  Set speed (76.2 mm/s)
  MoveL 645 to (-197.85, 148.44, -8.4) mm, rotated rx -174.06 ry -29.54 rz -11.91 deg; joints [4.931, -49.184, 110.878, -80.007, 60.979, 152.328]
  MoveL 646 to (-199.6, 148.44, -8.41) mm, rotated rx -174.06 ry -29.54 rz -11.91 deg; joints [4.86, -49.19, 110.892, -80.07, 60.944, 152.33]
  MoveL 647 to (-206.05, 148.44, -11.57) mm, rotated rx -174.06 ry -29.54 rz -11.91 deg; joints [4.602, -49.043, 110.941, -80.393, 60.791, 152.527]
  MoveL 648 to (-201.08, 148.44, -20.25) mm, rotated rx -174.06 ry -29.54 rz -11.91 deg; joints [4.803, -48.562, 110.904, -80.469, 60.81, 153.047]
  MoveL 649 to (-201.08, 145.27, -20.25) mm, rotated rx -174.06 ry -29.54 rz -11.91 deg; joints [4.814, -48.698, 111.183, -80.539, 60.791, 153.21]
  MoveL 650 to (-206.05, 145.27, -11.57) mm, rotated rx -174.06 ry -29.54 rz -11.91 deg; joints [4.613, -49.18, 111.22, -80.463, 60.772, 152.689]
  MoveL 651 to (-199.6, 145.27, -8.41) mm, rotated rx -174.06 ry -29.54 rz -11.91 deg; joints [4.872, -49.327, 111.171, -80.138, 60.925, 152.491]
  MoveL 652 to (-197.85, 145.27, -8.4) mm, rotated rx -174.06 ry -29.54 rz -11.91 deg; joints [4.942, -49.321, 111.158, -80.075, 60.959, 152.489]
  MoveL 653 to (-197.85, 145.27, -4.14) mm, rotated rx -174.06 ry -29.54 rz -11.91 deg; joints [4.941, -49.548, 111.154, -79.95, 60.999, 152.23]
  Set speed (38.1 mm/s)
  MoveL 654 to (-197.89, 145.27, -3.98) mm, rotated rx -174.06 ry -29.54 rz -11.91 deg; joints [4.939, -49.557, 111.155, -79.947, 60.999, 152.22]
  MoveL 655 to (-198.05, 144.95, -3.7) mm, rotated rx -174.06 ry -29.54 rz -11.91 deg; joints [4.934, -49.585, 111.183, -79.951, 60.997, 152.22]
  Set speed (76.2 mm/s)
  MoveL 656 to (-198.05, 142.41, -3.7) mm, rotated rx -174.06 ry -29.54 rz -11.91 deg; joints [4.943, -49.696, 111.406, -80.005, 60.981, 152.347]
  Set speed (38.1 mm/s)
  MoveL 657 to (-197.89, 142.09, -3.98) mm, rotated rx -174.06 ry -29.54 rz -11.91 deg; joints [4.951, -49.694, 111.433, -80.014, 60.98, 152.38]
  MoveL 658 to (-197.85, 142.09, -4.14) mm, rotated rx -174.06 ry -29.54 rz -11.91 deg; joints [4.952, -49.686, 111.433, -80.017, 60.979, 152.39]
  Set speed (76.2 mm/s)
  MoveL 659 to (-197.85, 142.09, -8.4) mm, rotated rx -174.06 ry -29.54 rz -11.91 deg; joints [4.953, -49.458, 111.436, -80.143, 60.94, 152.65]
  MoveL 660 to (-199.6, 142.09, -8.41) mm, rotated rx -174.06 ry -29.54 rz -11.91 deg; joints [4.883, -49.464, 111.45, -80.206, 60.906, 152.652]
  MoveL 661 to (-206.05, 142.09, -11.57) mm, rotated rx -174.06 ry -29.54 rz -11.91 deg; joints [4.623, -49.316, 111.499, -80.533, 60.753, 152.851]
  MoveL 662 to (-201.08, 142.09, -20.25) mm, rotated rx -174.06 ry -29.54 rz -11.91 deg; joints [4.825, -48.833, 111.462, -80.609, 60.773, 153.374]
  MoveL 663 to (-201.08, 138.92, -20.25) mm, rotated rx -174.06 ry -29.54 rz -11.91 deg; joints [4.836, -48.967, 111.74, -80.678, 60.754, 153.537]
  MoveL 664 to (-206.05, 138.92, -11.57) mm, rotated rx -174.06 ry -29.54 rz -11.91 deg; joints [4.634, -49.453, 111.777, -80.602, 60.735, 153.012]
  MoveL 665 to (-199.6, 138.92, -8.41) mm, rotated rx -174.06 ry -29.54 rz -11.91 deg; joints [4.894, -49.6, 111.728, -80.275, 60.887, 152.813]
  MoveL 666 to (-197.85, 138.92, -8.4) mm, rotated rx -174.06 ry -29.54 rz -11.91 deg; joints [4.965, -49.595, 111.714, -80.211, 60.921, 152.81]
  MoveL 667 to (-197.85, 138.92, -4.14) mm, rotated rx -174.06 ry -29.54 rz -11.91 deg; joints [4.964, -49.823, 111.711, -80.085, 60.96, 152.549]
  Set speed (38.1 mm/s)
  MoveL 668 to (-197.89, 138.92, -3.98) mm, rotated rx -174.06 ry -29.54 rz -11.91 deg; joints [4.962, -49.832, 111.711, -80.082, 60.961, 152.54]
  MoveL 669 to (-198.05, 138.6, -3.7) mm, rotated rx -174.06 ry -29.54 rz -11.91 deg; joints [4.957, -49.861, 111.74, -80.086, 60.959, 152.539]
  Set speed (76.2 mm/s)
  MoveL 670 to (-198.05, 136.06, -3.7) mm, rotated rx -174.06 ry -29.54 rz -11.91 deg; joints [4.966, -49.97, 111.962, -80.14, 60.944, 152.666]
  Set speed (38.1 mm/s)
  MoveL 671 to (-197.89, 135.74, -3.98) mm, rotated rx -174.06 ry -29.54 rz -11.91 deg; joints [4.973, -49.969, 111.989, -80.149, 60.942, 152.699]
  MoveL 672 to (-197.85, 135.74, -4.14) mm, rotated rx -174.06 ry -29.54 rz -11.91 deg; joints [4.975, -49.96, 111.988, -80.152, 60.942, 152.709]
  Set speed (76.2 mm/s)
  MoveL 673 to (-197.85, 135.74, -8.4) mm, rotated rx -174.06 ry -29.54 rz -11.91 deg; joints [4.976, -49.731, 111.992, -80.279, 60.903, 152.971]
  MoveL 674 to (-199.6, 135.74, -8.41) mm, rotated rx -174.06 ry -29.54 rz -11.91 deg; joints [4.905, -49.737, 112.005, -80.343, 60.869, 152.973]
  MoveL 675 to (-206.05, 135.74, -11.57) mm, rotated rx -174.06 ry -29.54 rz -11.91 deg; joints [4.644, -49.588, 112.055, -80.671, 60.717, 153.173]
  MoveL 676 to (-201.08, 135.74, -20.25) mm, rotated rx -174.06 ry -29.54 rz -11.91 deg; joints [4.848, -49.102, 112.018, -80.748, 60.736, 153.699]
  MoveL 677 to (-201.08, 132.57, -20.25) mm, rotated rx -174.06 ry -29.54 rz -11.91 deg; joints [4.859, -49.236, 112.295, -80.818, 60.718, 153.862]
  MoveL 678 to (-206.05, 132.57, -11.57) mm, rotated rx -174.06 ry -29.54 rz -11.91 deg; joints [4.655, -49.724, 112.332, -80.741, 60.699, 153.334]
  MoveL 679 to (-199.6, 132.57, -8.41) mm, rotated rx -174.06 ry -29.54 rz -11.91 deg; joints [4.916, -49.873, 112.282, -80.411, 60.85, 153.133]
  MoveL 680 to (-197.85, 132.57, -8.4) mm, rotated rx -174.06 ry -29.54 rz -11.91 deg; joints [4.987, -49.867, 112.269, -80.346, 60.884, 153.13]
  MoveL 681 to (-197.85, 132.57, -4.14) mm, rotated rx -174.06 ry -29.54 rz -11.91 deg; joints [4.987, -50.097, 112.265, -80.219, 60.923, 152.868]
  Set speed (38.1 mm/s)
  MoveL 682 to (-197.89, 132.57, -3.98) mm, rotated rx -174.06 ry -29.54 rz -11.91 deg; joints [4.985, -50.105, 112.266, -80.216, 60.924, 152.858]
  MoveL 683 to (-198.05, 132.25, -3.7) mm, rotated rx -174.06 ry -29.54 rz -11.91 deg; joints [4.979, -50.135, 112.294, -80.22, 60.921, 152.857]
  Set speed (76.2 mm/s)
  MoveL 684 to (-198.05, 129.71, -3.7) mm, rotated rx -174.06 ry -29.54 rz -11.91 deg; joints [4.989, -50.244, 112.515, -80.274, 60.906, 152.984]
  Set speed (38.1 mm/s)
  MoveL 685 to (-197.89, 129.39, -3.98) mm, rotated rx -174.06 ry -29.54 rz -11.91 deg; joints [4.996, -50.242, 112.542, -80.283, 60.905, 153.017]
  MoveL 686 to (-197.85, 129.39, -4.14) mm, rotated rx -174.06 ry -29.54 rz -11.91 deg; joints [4.998, -50.233, 112.542, -80.286, 60.905, 153.026]
  Set speed (76.2 mm/s)
  MoveL 687 to (-197.85, 129.39, -8.4) mm, rotated rx -174.06 ry -29.54 rz -11.91 deg; joints [4.999, -50.003, 112.545, -80.414, 60.866, 153.29]
  MoveL 688 to (-199.6, 129.39, -8.41) mm, rotated rx -174.06 ry -29.54 rz -11.91 deg; joints [4.928, -50.009, 112.559, -80.478, 60.832, 153.293]
  MoveL 689 to (-206.05, 129.39, -11.57) mm, rotated rx -174.06 ry -29.54 rz -11.91 deg; joints [4.666, -49.859, 112.608, -80.81, 60.681, 153.495]
  MoveL 690 to (-201.08, 129.39, -20.25) mm, rotated rx -174.06 ry -29.54 rz -11.91 deg; joints [4.87, -49.37, 112.571, -80.887, 60.701, 154.024]
  MoveL 691 to (-201.08, 126.22, -20.25) mm, rotated rx -174.06 ry -29.54 rz -11.91 deg; joints [4.881, -49.504, 112.847, -80.956, 60.683, 154.186]
  MoveL 692 to (-206.05, 126.22, -11.57) mm, rotated rx -174.06 ry -29.54 rz -11.91 deg; joints [4.677, -49.994, 112.884, -80.879, 60.664, 153.655]
  MoveL 693 to (-199.6, 126.22, -8.41) mm, rotated rx -174.06 ry -29.54 rz -11.91 deg; joints [4.939, -50.144, 112.834, -80.546, 60.814, 153.452]
  MoveL 694 to (-197.85, 126.22, -8.4) mm, rotated rx -174.06 ry -29.54 rz -11.91 deg; joints [5.01, -50.138, 112.821, -80.481, 60.848, 153.45]
  MoveL 695 to (-197.85, 126.22, -4.14) mm, rotated rx -174.06 ry -29.54 rz -11.91 deg; joints [5.01, -50.37, 112.818, -80.353, 60.886, 153.185]
  Set speed (38.1 mm/s)
  MoveL 696 to (-197.89, 126.22, -3.98) mm, rotated rx -174.06 ry -29.54 rz -11.91 deg; joints [5.008, -50.378, 112.818, -80.35, 60.887, 153.175]
  MoveL 697 to (-198.05, 125.9, -3.7) mm, rotated rx -174.06 ry -29.54 rz -11.91 deg; joints [5.002, -50.407, 112.846, -80.354, 60.885, 153.174]
  Set speed (76.2 mm/s)
  MoveL 698 to (-198.05, 123.36, -3.7) mm, rotated rx -174.06 ry -29.54 rz -11.91 deg; joints [5.012, -50.516, 113.067, -80.408, 60.87, 153.301]
  Set speed (38.1 mm/s)
  MoveL 699 to (-197.89, 123.04, -3.98) mm, rotated rx -174.06 ry -29.54 rz -11.91 deg; joints [5.019, -50.514, 113.093, -80.417, 60.869, 153.333]
  MoveL 700 to (-197.85, 123.04, -4.14) mm, rotated rx -174.06 ry -29.54 rz -11.91 deg; joints [5.021, -50.506, 113.093, -80.42, 60.868, 153.343]
  Set speed (76.2 mm/s)
  MoveL 701 to (-197.85, 123.04, -8.4) mm, rotated rx -174.06 ry -29.54 rz -11.91 deg; joints [5.022, -50.274, 113.096, -80.549, 60.83, 153.609]
  MoveL 702 to (-199.6, 123.04, -8.41) mm, rotated rx -174.06 ry -29.54 rz -11.91 deg; joints [4.95, -50.28, 113.11, -80.614, 60.796, 153.611]
  MoveL 703 to (-206.05, 123.04, -11.57) mm, rotated rx -174.06 ry -29.54 rz -11.91 deg; joints [4.687, -50.129, 113.159, -80.948, 60.646, 153.816]
  MoveL 704 to (-201.08, 123.04, -20.25) mm, rotated rx -174.06 ry -29.54 rz -11.91 deg; joints [4.892, -49.637, 113.122, -81.025, 60.666, 154.348]
  MoveL 705 to (-201.08, 119.87, -20.25) mm, rotated rx -174.06 ry -29.54 rz -11.91 deg; joints [4.904, -49.77, 113.397, -81.094, 60.649, 154.509]
  MoveL 706 to (-206.05, 119.87, -11.57) mm, rotated rx -174.06 ry -29.54 rz -11.91 deg; joints [4.698, -50.264, 113.434, -81.016, 60.629, 153.975]
  MoveL 707 to (-199.6, 119.87, -8.41) mm, rotated rx -174.06 ry -29.54 rz -11.91 deg; joints [4.962, -50.415, 113.385, -80.681, 60.779, 153.77]
  MoveL 708 to (-197.85, 119.87, -8.4) mm, rotated rx -174.06 ry -29.54 rz -11.91 deg; joints [5.034, -50.409, 113.371, -80.616, 60.812, 153.768]
  MoveL 709 to (-197.85, 119.87, -4.14) mm, rotated rx -174.06 ry -29.54 rz -11.91 deg; joints [5.033, -50.641, 113.368, -80.487, 60.851, 153.501]
  Set speed (38.1 mm/s)
  MoveL 710 to (-197.89, 119.87, -3.98) mm, rotated rx -174.06 ry -29.54 rz -11.91 deg; joints [5.031, -50.65, 113.368, -80.483, 60.851, 153.491]
  MoveL 711 to (-198.05, 119.55, -3.7) mm, rotated rx -174.06 ry -29.54 rz -11.91 deg; joints [5.026, -50.679, 113.396, -80.488, 60.849, 153.49]
  Set speed (76.2 mm/s)
  MoveL 712 to (-198.05, 117.01, -3.7) mm, rotated rx -174.06 ry -29.54 rz -11.91 deg; joints [5.035, -50.788, 113.616, -80.541, 60.835, 153.616]
  Set speed (38.1 mm/s)
  MoveL 713 to (-197.89, 116.7, -3.98) mm, rotated rx -174.06 ry -29.54 rz -11.91 deg; joints [5.043, -50.786, 113.642, -80.55, 60.834, 153.649]
  MoveL 714 to (-197.85, 116.7, -4.14) mm, rotated rx -174.06 ry -29.54 rz -11.91 deg; joints [5.044, -50.777, 113.642, -80.553, 60.833, 153.659]
  Set speed (76.2 mm/s)
  MoveL 715 to (-197.85, 116.7, -8.4) mm, rotated rx -174.06 ry -29.54 rz -11.91 deg; joints [5.045, -50.543, 113.645, -80.683, 60.795, 153.926]
  MoveL 716 to (-199.6, 116.7, -8.41) mm, rotated rx -174.06 ry -29.54 rz -11.91 deg; joints [4.973, -50.549, 113.659, -80.748, 60.761, 153.929]
  MoveL 717 to (-206.05, 116.7, -11.57) mm, rotated rx -174.06 ry -29.54 rz -11.91 deg; joints [4.709, -50.398, 113.708, -81.085, 60.612, 154.135]
  MoveL 718 to (-201.08, 116.7, -20.25) mm, rotated rx -174.06 ry -29.54 rz -11.91 deg; joints [4.915, -49.903, 113.671, -81.163, 60.632, 154.671]
  MoveL 719 to (-201.08, 113.52, -20.25) mm, rotated rx -174.06 ry -29.54 rz -11.91 deg; joints [4.927, -50.035, 113.945, -81.232, 60.615, 154.832]
  MoveL 720 to (-206.05, 113.52, -11.57) mm, rotated rx -174.06 ry -29.54 rz -11.91 deg; joints [4.72, -50.532, 113.982, -81.153, 60.595, 154.295]
  MoveL 721 to (-199.6, 113.52, -8.41) mm, rotated rx -174.06 ry -29.54 rz -11.91 deg; joints [4.985, -50.684, 113.933, -80.815, 60.744, 154.088]
  MoveL 722 to (-197.85, 113.52, -8.4) mm, rotated rx -174.06 ry -29.54 rz -11.91 deg; joints [5.057, -50.678, 113.919, -80.75, 60.778, 154.085]
  MoveL 723 to (-197.85, 113.52, -4.14) mm, rotated rx -174.06 ry -29.54 rz -11.91 deg; joints [5.056, -50.912, 113.916, -80.62, 60.816, 153.817]
  Set speed (38.1 mm/s)
  MoveL 724 to (-197.89, 113.52, -3.98) mm, rotated rx -174.06 ry -29.54 rz -11.91 deg; joints [5.054, -50.921, 113.916, -80.616, 60.816, 153.807]
  MoveL 725 to (-198.05, 113.2, -3.7) mm, rotated rx -174.06 ry -29.54 rz -11.91 deg; joints [5.049, -50.95, 113.944, -80.62, 60.814, 153.805]
  Set speed (76.2 mm/s)
  MoveL 726 to (-198.05, 110.66, -3.7) mm, rotated rx -174.06 ry -29.54 rz -11.91 deg; joints [5.058, -51.058, 114.163, -80.673, 60.8, 153.931]
  Set speed (38.1 mm/s)
  MoveL 727 to (-197.89, 110.35, -3.98) mm, rotated rx -174.06 ry -29.54 rz -11.91 deg; joints [5.066, -51.056, 114.189, -80.682, 60.799, 153.964]
  MoveL 728 to (-197.85, 110.35, -4.14) mm, rotated rx -174.06 ry -29.54 rz -11.91 deg; joints [5.068, -51.047, 114.189, -80.686, 60.798, 153.974]
  Set speed (76.2 mm/s)
  MoveL 729 to (-197.85, 110.35, -8.4) mm, rotated rx -174.06 ry -29.54 rz -11.91 deg; joints [5.069, -50.812, 114.192, -80.816, 60.761, 154.243]
  MoveL 730 to (-199.6, 110.35, -8.41) mm, rotated rx -174.06 ry -29.54 rz -11.91 deg; joints [4.997, -50.818, 114.206, -80.882, 60.727, 154.246]
  MoveL 731 to (-206.05, 110.35, -11.57) mm, rotated rx -174.06 ry -29.54 rz -11.91 deg; joints [4.731, -50.665, 114.255, -81.222, 60.579, 154.454]
  MoveL 732 to (-201.08, 110.35, -20.25) mm, rotated rx -174.06 ry -29.54 rz -11.91 deg; joints [4.938, -50.167, 114.218, -81.301, 60.599, 154.993]
  MoveL 733 to (-201.08, 107.17, -20.25) mm, rotated rx -174.06 ry -29.54 rz -11.91 deg; joints [4.95, -50.299, 114.491, -81.369, 60.583, 155.153]
  MoveL 734 to (-206.05, 107.17, -11.57) mm, rotated rx -174.06 ry -29.54 rz -11.91 deg; joints [4.742, -50.799, 114.528, -81.29, 60.563, 154.613]
  MoveL 735 to (-199.6, 107.17, -8.41) mm, rotated rx -174.06 ry -29.54 rz -11.91 deg; joints [5.008, -50.952, 114.479, -80.949, 60.711, 154.404]
  MoveL 736 to (-197.85, 107.17, -8.4) mm, rotated rx -174.06 ry -29.54 rz -11.91 deg; joints [5.081, -50.946, 114.465, -80.883, 60.744, 154.401]
  MoveL 737 to (-197.85, 107.17, -4.14) mm, rotated rx -174.06 ry -29.54 rz -11.91 deg; joints [5.08, -51.181, 114.462, -80.752, 60.781, 154.131]
  Set speed (38.1 mm/s)
  MoveL 738 to (-197.89, 107.17, -3.98) mm, rotated rx -174.06 ry -29.54 rz -11.91 deg; joints [5.078, -51.19, 114.462, -80.749, 60.782, 154.121]
  MoveL 739 to (-198.05, 106.85, -3.7) mm, rotated rx -174.06 ry -29.54 rz -11.91 deg; joints [5.073, -51.22, 114.49, -80.753, 60.78, 154.12]
  Set speed (76.2 mm/s)
  MoveL 740 to (-198.05, 104.31, -3.7) mm, rotated rx -174.06 ry -29.54 rz -11.91 deg; joints [5.082, -51.327, 114.708, -80.805, 60.766, 154.245]
  Set speed (38.1 mm/s)
  MoveL 741 to (-197.89, 104, -3.98) mm, rotated rx -174.06 ry -29.54 rz -11.91 deg; joints [5.09, -51.325, 114.734, -80.814, 60.765, 154.278]
  MoveL 742 to (-197.85, 104, -4.14) mm, rotated rx -174.06 ry -29.54 rz -11.91 deg; joints [5.092, -51.316, 114.734, -80.818, 60.765, 154.288]
  Set speed (76.2 mm/s)
  MoveL 743 to (-197.85, 104, -8.4) mm, rotated rx -174.06 ry -29.54 rz -11.91 deg; joints [5.093, -51.08, 114.737, -80.949, 60.727, 154.559]
  MoveL 744 to (-199.6, 104, -8.41) mm, rotated rx -174.06 ry -29.54 rz -11.91 deg; joints [5.02, -51.086, 114.751, -81.016, 60.694, 154.562]
  MoveL 745 to (-206.05, 104, -11.57) mm, rotated rx -174.06 ry -29.54 rz -11.91 deg; joints [4.753, -50.932, 114.801, -81.358, 60.546, 154.772]
  MoveL 746 to (-201.08, 104, -20.25) mm, rotated rx -174.06 ry -29.54 rz -11.91 deg; joints [4.961, -50.431, 114.763, -81.438, 60.567, 155.314]
  MoveL 747 to (-201.08, 100.82, -20.25) mm, rotated rx -174.06 ry -29.54 rz -11.91 deg; joints [4.973, -50.562, 115.035, -81.506, 60.551, 155.474]
  MoveL 748 to (-206.05, 100.82, -11.57) mm, rotated rx -174.06 ry -29.54 rz -11.91 deg; joints [4.765, -51.065, 115.072, -81.426, 60.53, 154.93]
  MoveL 749 to (-199.6, 100.82, -8.41) mm, rotated rx -174.06 ry -29.54 rz -11.91 deg; joints [5.032, -51.219, 115.023, -81.082, 60.678, 154.72]
  MoveL 750 to (-197.85, 100.82, -8.4) mm, rotated rx -174.06 ry -29.54 rz -11.91 deg; joints [5.105, -51.213, 115.009, -81.016, 60.711, 154.716]
  MoveL 751 to (-197.85, 100.82, -4.14) mm, rotated rx -174.06 ry -29.54 rz -11.91 deg; joints [5.104, -51.45, 115.006, -80.884, 60.748, 154.445]
  Set speed (38.1 mm/s)
  MoveL 752 to (-197.89, 100.82, -3.98) mm, rotated rx -174.06 ry -29.54 rz -11.91 deg; joints [5.102, -51.459, 115.006, -80.88, 60.749, 154.434]
  MoveL 753 to (-198.05, 100.5, -3.7) mm, rotated rx -174.06 ry -29.54 rz -11.91 deg; joints [5.096, -51.488, 115.034, -80.884, 60.746, 154.433]
  Set speed (76.2 mm/s)
  MoveL 754 to (-198.05, 97.96, -3.7) mm, rotated rx -174.06 ry -29.54 rz -11.91 deg; joints [5.106, -51.595, 115.251, -80.937, 60.733, 154.558]
  Set speed (38.1 mm/s)
  MoveL 755 to (-197.89, 97.65, -3.98) mm, rotated rx -174.06 ry -29.54 rz -11.91 deg; joints [5.114, -51.593, 115.277, -80.946, 60.732, 154.591]
  MoveL 756 to (-197.85, 97.65, -4.14) mm, rotated rx -174.06 ry -29.54 rz -11.91 deg; joints [5.116, -51.584, 115.277, -80.949, 60.732, 154.601]
  Set speed (76.2 mm/s)
  MoveL 757 to (-197.85, 97.65, -8.4) mm, rotated rx -174.06 ry -29.54 rz -11.91 deg; joints [5.117, -51.346, 115.28, -81.082, 60.694, 154.874]
  MoveL 758 to (-199.6, 97.65, -8.41) mm, rotated rx -174.06 ry -29.54 rz -11.91 deg; joints [5.044, -51.352, 115.294, -81.149, 60.661, 154.877]
  MoveL 759 to (-206.05, 97.65, -11.57) mm, rotated rx -174.06 ry -29.54 rz -11.91 deg; joints [4.776, -51.197, 115.344, -81.494, 60.515, 155.088]
  MoveL 760 to (-201.08, 97.65, -20.25) mm, rotated rx -174.06 ry -29.54 rz -11.91 deg; joints [4.985, -50.693, 115.306, -81.574, 60.535, 155.634]
  MoveL 761 to (-201.08, 94.47, -20.25) mm, rotated rx -174.06 ry -29.54 rz -11.91 deg; joints [4.996, -50.824, 115.577, -81.642, 60.52, 155.794]
  MoveL 762 to (-206.05, 94.47, -11.57) mm, rotated rx -174.06 ry -29.54 rz -11.91 deg; joints [4.787, -51.33, 115.614, -81.561, 60.499, 155.247]
  MoveL 763 to (-199.6, 94.47, -8.41) mm, rotated rx -174.06 ry -29.54 rz -11.91 deg; joints [5.056, -51.485, 115.565, -81.215, 60.645, 155.034]
  MoveL 764 to (-197.85, 94.47, -8.4) mm, rotated rx -174.06 ry -29.54 rz -11.91 deg; joints [5.129, -51.479, 115.551, -81.148, 60.678, 155.031]
  MoveL 765 to (-197.85, 94.47, -4.14) mm, rotated rx -174.06 ry -29.54 rz -11.91 deg; joints [5.128, -51.718, 115.548, -81.015, 60.715, 154.757]
  Set speed (38.1 mm/s)
  MoveL 766 to (-197.89, 94.47, -3.98) mm, rotated rx -174.06 ry -29.54 rz -11.91 deg; joints [5.126, -51.727, 115.548, -81.011, 60.716, 154.747]
  MoveL 767 to (-198.05, 94.15, -3.7) mm, rotated rx -174.06 ry -29.54 rz -11.91 deg; joints [5.12, -51.756, 115.576, -81.016, 60.714, 154.745]
  Set speed (76.2 mm/s)
  MoveL 768 to (-198.05, 91.61, -3.7) mm, rotated rx -174.06 ry -29.54 rz -11.91 deg; joints [5.13, -51.863, 115.792, -81.068, 60.701, 154.87]
  Set speed (38.1 mm/s)
  MoveL 769 to (-197.89, 91.3, -3.98) mm, rotated rx -174.06 ry -29.54 rz -11.91 deg; joints [5.138, -51.86, 115.818, -81.077, 60.7, 154.903]
  MoveL 770 to (-197.85, 91.3, -4.14) mm, rotated rx -174.06 ry -29.54 rz -11.91 deg; joints [5.14, -51.851, 115.818, -81.08, 60.699, 154.913]
  Set speed (76.2 mm/s)
  MoveL 771 to (-197.85, 91.3, -8.4) mm, rotated rx -174.06 ry -29.54 rz -11.91 deg; joints [5.141, -51.612, 115.821, -81.214, 60.662, 155.188]
  MoveL 772 to (-200.08, 91.3, -8.41) mm, rotated rx -174.06 ry -29.54 rz -11.91 deg; joints [5.047, -51.619, 115.839, -81.3, 60.621, 155.192]
  MoveL 773 to (-206.05, 91.3, -11.57) mm, rotated rx -174.06 ry -29.54 rz -11.91 deg; joints [4.798, -51.462, 115.885, -81.629, 60.484, 155.404]
  MoveL 774 to (-201.08, 91.3, -20.25) mm, rotated rx -174.06 ry -29.54 rz -11.91 deg; joints [5.008, -50.955, 115.847, -81.71, 60.505, 155.954]
  MoveL 775 to (-201.08, 88.12, -20.25) mm, rotated rx -174.06 ry -29.54 rz -11.91 deg; joints [5.02, -51.085, 116.117, -81.778, 60.49, 156.113]
  MoveL 776 to (-206.05, 88.12, -11.57) mm, rotated rx -174.06 ry -29.54 rz -11.91 deg; joints [4.81, -51.594, 116.154, -81.696, 60.469, 155.562]
  MoveL 777 to (-200.08, 88.12, -8.41) mm, rotated rx -174.06 ry -29.54 rz -11.91 deg; joints [5.059, -51.752, 116.108, -81.366, 60.605, 155.349]
  MoveL 778 to (-197.85, 88.12, -8.4) mm, rotated rx -174.06 ry -29.54 rz -11.91 deg; joints [5.153, -51.744, 116.091, -81.28, 60.647, 155.344]
  MoveL 779 to (-197.85, 88.12, -4.14) mm, rotated rx -174.06 ry -29.54 rz -11.91 deg; joints [5.152, -51.984, 116.088, -81.146, 60.683, 155.069]
  Set speed (38.1 mm/s)
  MoveL 780 to (-197.89, 88.12, -3.98) mm, rotated rx -174.06 ry -29.54 rz -11.91 deg; joints [5.15, -51.993, 116.088, -81.142, 60.684, 155.059]
  MoveL 781 to (-198.05, 87.81, -3.7) mm, rotated rx -174.06 ry -29.54 rz -11.91 deg; joints [5.145, -52.022, 116.116, -81.146, 60.682, 155.057]
  Set speed (76.2 mm/s)
  MoveL 782 to (-198.05, 85.27, -3.7) mm, rotated rx -174.06 ry -29.54 rz -11.91 deg; joints [5.154, -52.129, 116.331, -81.198, 60.669, 155.181]
  Set speed (38.1 mm/s)
  MoveL 783 to (-197.89, 84.95, -3.98) mm, rotated rx -174.06 ry -29.54 rz -11.91 deg; joints [5.162, -52.126, 116.357, -81.207, 60.668, 155.214]
  MoveL 784 to (-197.85, 84.95, -4.14) mm, rotated rx -174.06 ry -29.54 rz -11.91 deg; joints [5.164, -52.117, 116.357, -81.211, 60.668, 155.224]
  Set speed (76.2 mm/s)
  MoveL 785 to (-197.85, 84.95, -8.4) mm, rotated rx -174.06 ry -29.54 rz -11.91 deg; joints [5.165, -51.876, 116.36, -81.345, 60.631, 155.501]
  MoveL 786 to (-200.08, 84.95, -8.41) mm, rotated rx -174.06 ry -29.54 rz -11.91 deg; joints [5.071, -51.884, 116.378, -81.432, 60.59, 155.505]
  MoveL 787 to (-206.05, 84.95, -11.57) mm, rotated rx -174.06 ry -29.54 rz -11.91 deg; joints [4.821, -51.725, 116.424, -81.764, 60.454, 155.72]
  MoveL 788 to (-201.08, 84.95, -20.25) mm, rotated rx -174.06 ry -29.54 rz -11.91 deg; joints [5.032, -51.215, 116.386, -81.845, 60.475, 156.272]
  MoveL 789 to (-201.08, 81.77, -20.25) mm, rotated rx -174.06 ry -29.54 rz -11.91 deg; joints [5.044, -51.345, 116.655, -81.913, 60.46, 156.431]
  MoveL 790 to (-206.05, 81.77, -11.57) mm, rotated rx -174.06 ry -29.54 rz -11.91 deg; joints [4.833, -51.857, 116.692, -81.831, 60.439, 155.877]
  MoveL 791 to (-200.08, 81.77, -8.41) mm, rotated rx -174.06 ry -29.54 rz -11.91 deg; joints [5.083, -52.016, 116.646, -81.498, 60.575, 155.661]
  MoveL 792 to (-197.85, 81.77, -8.4) mm, rotated rx -174.06 ry -29.54 rz -11.91 deg; joints [5.178, -52.008, 116.629, -81.411, 60.616, 155.657]
  MoveL 793 to (-197.85, 81.77, -4.14) mm, rotated rx -174.06 ry -29.54 rz -11.91 deg; joints [5.177, -52.25, 116.626, -81.276, 60.652, 155.38]
  Set speed (38.1 mm/s)
  MoveL 794 to (-197.89, 81.77, -3.98) mm, rotated rx -174.06 ry -29.54 rz -11.91 deg; joints [5.175, -52.259, 116.626, -81.272, 60.653, 155.369]
  MoveL 795 to (-198.05, 81.46, -3.7) mm, rotated rx -174.06 ry -29.54 rz -11.91 deg; joints [5.169, -52.288, 116.654, -81.276, 60.651, 155.367]
  Set speed (76.2 mm/s)
  MoveL 796 to (-198.05, 78.92, -3.7) mm, rotated rx -174.06 ry -29.54 rz -11.91 deg; joints [5.179, -52.394, 116.868, -81.328, 60.639, 155.491]
  Set speed (38.1 mm/s)
  MoveL 797 to (-197.89, 78.6, -3.98) mm, rotated rx -174.06 ry -29.54 rz -11.91 deg; joints [5.187, -52.391, 116.894, -81.337, 60.638, 155.524]
  MoveL 798 to (-197.85, 78.6, -4.14) mm, rotated rx -174.06 ry -29.54 rz -11.91 deg; joints [5.189, -52.382, 116.894, -81.341, 60.637, 155.535]
  Set speed (76.2 mm/s)
  MoveL 799 to (-197.85, 78.6, -8.4) mm, rotated rx -174.06 ry -29.54 rz -11.91 deg; joints [5.19, -52.14, 116.897, -81.476, 60.601, 155.813]
  MoveL 800 to (-200.08, 78.6, -8.41) mm, rotated rx -174.06 ry -29.54 rz -11.91 deg; joints [5.095, -52.147, 116.915, -81.564, 60.56, 155.817]
  MoveL 801 to (-206.05, 78.6, -11.57) mm, rotated rx -174.06 ry -29.54 rz -11.91 deg; joints [4.844, -51.988, 116.961, -81.898, 60.424, 156.034]
  MoveL 802 to (-201.08, 78.6, -20.25) mm, rotated rx -174.06 ry -29.54 rz -11.91 deg; joints [5.056, -51.474, 116.923, -81.98, 60.446, 156.59]
  MoveL 803 to (-201.08, 75.42, -20.25) mm, rotated rx -174.06 ry -29.54 rz -11.91 deg; joints [5.068, -51.604, 117.191, -82.047, 60.431, 156.749]
  MoveL 804 to (-206.05, 75.42, -11.57) mm, rotated rx -174.06 ry -29.54 rz -11.91 deg; joints [4.856, -52.119, 117.229, -81.965, 60.41, 156.191]
  MoveL 805 to (-200.08, 75.42, -8.41) mm, rotated rx -174.06 ry -29.54 rz -11.91 deg; joints [5.108, -52.279, 117.183, -81.629, 60.545, 155.973]
  MoveL 806 to (-197.85, 75.42, -8.4) mm, rotated rx -174.06 ry -29.54 rz -11.91 deg; joints [5.202, -52.271, 117.165, -81.542, 60.586, 155.969]
  MoveL 807 to (-197.85, 75.42, -4.14) mm, rotated rx -174.06 ry -29.54 rz -11.91 deg; joints [5.201, -52.514, 117.162, -81.405, 60.622, 155.689]
  Set speed (38.1 mm/s)
  MoveL 808 to (-197.89, 75.42, -3.98) mm, rotated rx -174.06 ry -29.54 rz -11.91 deg; joints [5.199, -52.523, 117.162, -81.402, 60.623, 155.679]
  MoveL 809 to (-198.05, 75.11, -3.7) mm, rotated rx -174.06 ry -29.54 rz -11.91 deg; joints [5.194, -52.553, 117.19, -81.406, 60.62, 155.677]
  Set speed (76.2 mm/s)
  MoveL 810 to (-198.05, 72.57, -3.7) mm, rotated rx -174.06 ry -29.54 rz -11.91 deg; joints [5.204, -52.658, 117.404, -81.457, 60.609, 155.8]
  Set speed (38.1 mm/s)
  MoveL 811 to (-197.89, 72.25, -3.98) mm, rotated rx -174.06 ry -29.54 rz -11.91 deg; joints [5.212, -52.655, 117.429, -81.466, 60.608, 155.834]
  MoveL 812 to (-197.85, 72.25, -4.14) mm, rotated rx -174.06 ry -29.54 rz -11.91 deg; joints [5.214, -52.646, 117.429, -81.47, 60.607, 155.844]
  Set speed (76.2 mm/s)
  MoveL 813 to (-197.85, 72.25, -8.4) mm, rotated rx -174.06 ry -29.54 rz -11.91 deg; joints [5.215, -52.403, 117.433, -81.607, 60.571, 156.125]
  MoveL 814 to (-200.08, 72.25, -8.41) mm, rotated rx -174.06 ry -29.54 rz -11.91 deg; joints [5.12, -52.41, 117.45, -81.695, 60.53, 156.129]
  MoveL 815 to (-206.05, 72.25, -11.57) mm, rotated rx -174.06 ry -29.54 rz -11.91 deg; joints [4.868, -52.249, 117.496, -82.031, 60.396, 156.347]
  MoveL 816 to (-201.08, 72.25, -20.25) mm, rotated rx -174.06 ry -29.54 rz -11.91 deg; joints [5.08, -51.733, 117.459, -82.114, 60.417, 156.907]
  MoveL 817 to (-201.08, 69.07, -20.25) mm, rotated rx -174.06 ry -29.54 rz -11.91 deg; joints [5.093, -51.862, 117.726, -82.181, 60.403, 157.065]
  MoveL 818 to (-206.05, 69.07, -11.57) mm, rotated rx -174.06 ry -29.54 rz -11.91 deg; joints [4.879, -52.38, 117.763, -82.098, 60.382, 156.504]
  MoveL 819 to (-200.08, 69.07, -8.41) mm, rotated rx -174.06 ry -29.54 rz -11.91 deg; joints [5.132, -52.541, 117.717, -81.76, 60.516, 156.284]
  MoveL 820 to (-197.85, 69.07, -8.4) mm, rotated rx -174.06 ry -29.54 rz -11.91 deg; joints [5.227, -52.533, 117.7, -81.672, 60.557, 156.28]
  MoveL 821 to (-197.85, 69.07, -4.14) mm, rotated rx -174.06 ry -29.54 rz -11.91 deg; joints [5.226, -52.778, 117.696, -81.534, 60.592, 155.998]
  Set speed (38.1 mm/s)
  MoveL 822 to (-197.89, 69.07, -3.98) mm, rotated rx -174.06 ry -29.54 rz -11.91 deg; joints [5.224, -52.787, 117.696, -81.531, 60.593, 155.988]
  MoveL 823 to (-198.05, 68.76, -3.7) mm, rotated rx -174.06 ry -29.54 rz -11.91 deg; joints [5.219, -52.817, 117.724, -81.535, 60.591, 155.986]
  Set speed (76.2 mm/s)
  MoveL 824 to (-198.05, 66.22, -3.7) mm, rotated rx -174.06 ry -29.54 rz -11.91 deg; joints [5.229, -52.922, 117.937, -81.586, 60.579, 156.109]
  Set speed (38.1 mm/s)
  MoveL 825 to (-197.89, 65.9, -3.98) mm, rotated rx -174.06 ry -29.54 rz -11.91 deg; joints [5.237, -52.919, 117.963, -81.595, 60.578, 156.142]
  MoveL 826 to (-197.85, 65.9, -4.14) mm, rotated rx -174.06 ry -29.54 rz -11.91 deg; joints [5.239, -52.909, 117.963, -81.599, 60.578, 156.153]
  Set speed (76.2 mm/s)
  MoveL 827 to (-197.85, 65.9, -8.4) mm, rotated rx -174.06 ry -29.54 rz -11.91 deg; joints [5.24, -52.664, 117.966, -81.737, 60.542, 156.435]
  MoveL 828 to (-200.08, 65.9, -8.41) mm, rotated rx -174.06 ry -29.54 rz -11.91 deg; joints [5.145, -52.672, 117.983, -81.825, 60.501, 156.44]
  MoveL 829 to (-206.05, 65.9, -11.57) mm, rotated rx -174.06 ry -29.54 rz -11.91 deg; joints [4.891, -52.51, 118.03, -82.165, 60.368, 156.66]
  MoveL 830 to (-201.08, 65.9, -20.25) mm, rotated rx -174.06 ry -29.54 rz -11.91 deg; joints [5.105, -51.99, 117.992, -82.248, 60.39, 157.223]
  MoveL 831 to (-201.08, 62.72, -20.25) mm, rotated rx -174.06 ry -29.54 rz -11.91 deg; joints [5.117, -52.118, 118.258, -82.315, 60.376, 157.381]
  MoveL 832 to (-206.05, 62.72, -11.57) mm, rotated rx -174.06 ry -29.54 rz -11.91 deg; joints [4.903, -52.64, 118.296, -82.231, 60.354, 156.816]
  MoveL 833 to (-200.08, 62.72, -8.41) mm, rotated rx -174.06 ry -29.54 rz -11.91 deg; joints [5.157, -52.802, 118.249, -81.891, 60.487, 156.595]
  MoveL 834 to (-197.85, 62.72, -8.4) mm, rotated rx -174.06 ry -29.54 rz -11.91 deg; joints [5.252, -52.795, 118.232, -81.801, 60.528, 156.59]
  MoveL 835 to (-197.85, 62.72, -4.14) mm, rotated rx -174.06 ry -29.54 rz -11.91 deg; joints [5.252, -53.041, 118.229, -81.663, 60.563, 156.307]
  Set speed (38.1 mm/s)
  MoveL 836 to (-197.89, 62.72, -3.98) mm, rotated rx -174.06 ry -29.54 rz -11.91 deg; joints [5.25, -53.05, 118.229, -81.659, 60.564, 156.296]
  MoveL 837 to (-198.05, 62.41, -3.7) mm, rotated rx -174.06 ry -29.54 rz -11.91 deg; joints [5.244, -53.079, 118.256, -81.663, 60.562, 156.293]
  Set speed (76.2 mm/s)
  MoveL 838 to (-198.05, 59.87, -3.7) mm, rotated rx -174.06 ry -29.54 rz -11.91 deg; joints [5.254, -53.184, 118.469, -81.714, 60.551, 156.416]
  Set speed (38.1 mm/s)
  MoveL 839 to (-197.89, 59.55, -3.98) mm, rotated rx -174.06 ry -29.54 rz -11.91 deg; joints [5.262, -53.181, 118.494, -81.723, 60.55, 156.45]
  MoveL 840 to (-197.85, 59.55, -4.14) mm, rotated rx -174.06 ry -29.54 rz -11.91 deg; joints [5.264, -53.172, 118.494, -81.727, 60.549, 156.46]
  Set speed (76.2 mm/s)
  MoveL 841 to (-197.85, 59.55, -8.4) mm, rotated rx -174.06 ry -29.54 rz -11.91 deg; joints [5.265, -52.925, 118.498, -81.866, 60.514, 156.745]
  MoveL 842 to (-200.08, 59.55, -8.41) mm, rotated rx -174.06 ry -29.54 rz -11.91 deg; joints [5.169, -52.932, 118.515, -81.955, 60.473, 156.75]
  MoveL 843 to (-206.05, 59.55, -11.57) mm, rotated rx -174.06 ry -29.54 rz -11.91 deg; joints [4.915, -52.769, 118.561, -82.297, 60.341, 156.972]
  MoveL 844 to (-201.08, 59.55, -20.25) mm, rotated rx -174.06 ry -29.54 rz -11.91 deg; joints [5.13, -52.246, 118.524, -82.381, 60.363, 157.539]
  MoveL 845 to (-201.08, 56.38, -20.25) mm, rotated rx -174.06 ry -29.54 rz -11.91 deg; joints [5.142, -52.374, 118.789, -82.448, 60.349, 157.696]
  MoveL 846 to (-206.05, 56.38, -11.57) mm, rotated rx -174.06 ry -29.54 rz -11.91 deg; joints [4.927, -52.899, 118.826, -82.363, 60.328, 157.127]
  MoveL 847 to (-200.08, 56.38, -8.41) mm, rotated rx -174.06 ry -29.54 rz -11.91 deg; joints [5.182, -53.062, 118.78, -82.02, 60.46, 156.904]
  MoveL 848 to (-197.85, 56.38, -8.4) mm, rotated rx -174.06 ry -29.54 rz -11.91 deg; joints [5.278, -53.055, 118.763, -81.93, 60.5, 156.899]
  MoveL 849 to (-197.85, 56.38, -4.14) mm, rotated rx -174.06 ry -29.54 rz -11.91 deg; joints [5.277, -53.302, 118.759, -81.791, 60.535, 156.614]
  Set speed (38.1 mm/s)
  MoveL 850 to (-197.89, 56.38, -3.98) mm, rotated rx -174.06 ry -29.54 rz -11.91 deg; joints [5.275, -53.312, 118.759, -81.787, 60.536, 156.603]
  MoveL 851 to (-198.05, 56.06, -3.7) mm, rotated rx -174.06 ry -29.54 rz -11.91 deg; joints [5.27, -53.341, 118.787, -81.791, 60.534, 156.601]
  Set speed (76.2 mm/s)
  MoveL 852 to (-198.05, 53.52, -3.7) mm, rotated rx -174.06 ry -29.54 rz -11.91 deg; joints [5.28, -53.446, 118.999, -81.842, 60.523, 156.723]
  Set speed (38.1 mm/s)
  MoveL 853 to (-197.89, 53.2, -3.98) mm, rotated rx -174.06 ry -29.54 rz -11.91 deg; joints [5.288, -53.442, 119.024, -81.851, 60.522, 156.757]
  MoveL 854 to (-197.85, 53.2, -4.14) mm, rotated rx -174.06 ry -29.54 rz -11.91 deg; joints [5.29, -53.433, 119.024, -81.855, 60.522, 156.767]
  Set speed (76.2 mm/s)
  MoveL 855 to (-197.85, 53.2, -8.4) mm, rotated rx -174.06 ry -29.54 rz -11.91 deg; joints [5.291, -53.185, 119.027, -81.995, 60.487, 157.054]
  MoveL 856 to (-200.08, 53.2, -8.41) mm, rotated rx -174.06 ry -29.54 rz -11.91 deg; joints [5.195, -53.192, 119.045, -82.085, 60.446, 157.059]
  MoveL 857 to (-206.05, 53.2, -11.57) mm, rotated rx -174.06 ry -29.54 rz -11.91 deg; joints [4.939, -53.028, 119.091, -82.429, 60.315, 157.283]
  MoveL 858 to (-201.08, 53.2, -20.25) mm, rotated rx -174.06 ry -29.54 rz -11.91 deg; joints [5.154, -52.502, 119.054, -82.514, 60.336, 157.853]
  MoveL 859 to (-201.08, 50.03, -20.25) mm, rotated rx -174.06 ry -29.54 rz -11.91 deg; joints [5.167, -52.629, 119.318, -82.58, 60.324, 158.01]
  MoveL 860 to (-206.05, 50.03, -11.57) mm, rotated rx -174.06 ry -29.54 rz -11.91 deg; joints [4.951, -53.157, 119.355, -82.495, 60.302, 157.438]
  MoveL 861 to (-200.08, 50.03, -8.41) mm, rotated rx -174.06 ry -29.54 rz -11.91 deg; joints [5.207, -53.322, 119.309, -82.149, 60.433, 157.213]
  MoveL 862 to (-197.85, 50.03, -8.4) mm, rotated rx -174.06 ry -29.54 rz -11.91 deg; joints [5.304, -53.314, 119.291, -82.059, 60.473, 157.208]
  MoveL 863 to (-197.85, 50.03, -4.14) mm, rotated rx -174.06 ry -29.54 rz -11.91 deg; joints [5.303, -53.563, 119.288, -81.918, 60.508, 156.92]
  Set speed (38.1 mm/s)
  MoveL 864 to (-197.89, 50.03, -3.98) mm, rotated rx -174.06 ry -29.54 rz -11.91 deg; joints [5.301, -53.573, 119.288, -81.915, 60.508, 156.91]
  MoveL 865 to (-197.93, 49.74, -3.64) mm, rotated rx -174.06 ry -29.54 rz -11.91 deg; joints [5.3, -53.605, 119.312, -81.911, 60.509, 156.901]
  Set speed (76.2 mm/s)
  MoveL 866 to (-196.9, 47.14, -3.04) mm, rotated rx -174.06 ry -29.54 rz -11.91 deg; joints [5.355, -53.743, 119.519, -81.901, 60.522, 156.983]
  Set speed (38.1 mm/s)
  MoveL 867 to (-196.62, 46.85, -3.25) mm, rotated rx -174.06 ry -29.54 rz -11.91 deg; joints [5.368, -53.741, 119.541, -81.903, 60.524, 157.01]
  MoveL 868 to (-195.49, 46.85, -5.2) mm, rotated rx -174.06 ry -29.54 rz -11.91 deg; joints [5.418, -53.623, 119.534, -81.922, 60.528, 157.14]
  MoveL 869 to (-195.45, 46.85, -5.36) mm, rotated rx -174.06 ry -29.54 rz -11.91 deg; joints [5.419, -53.613, 119.534, -81.925, 60.528, 157.151]
  Set speed (76.2 mm/s)
  MoveL 870 to (-195.45, 46.85, -9.71) mm, rotated rx -174.06 ry -29.54 rz -11.91 deg; joints [5.42, -53.358, 119.537, -82.069, 60.492, 157.444]
  MoveL 871 to (-203.6, 46.85, -10.15) mm, rotated rx -174.06 ry -29.54 rz -11.91 deg; joints [5.068, -53.361, 119.6, -82.414, 60.343, 157.492]
  MoveL 872 to (-198.68, 46.85, -18.86) mm, rotated rx -174.06 ry -29.54 rz -11.91 deg; joints [5.283, -52.83, 119.564, -82.503, 60.363, 158.068]
  Set speed (38.1 mm/s)
  MoveL 873 to (-199.55, 46.85, -18.63) mm, rotated rx -174.06 ry -29.54 rz -11.91 deg; joints [5.245, -52.847, 119.57, -82.531, 60.35, 158.055]
  Set speed (100.0 mm/s)
  MoveL 874 to (-233.61, 46.85, 40.17) mm, rotated rx -174.06 ry -29.54 rz -11.91 deg; joints [3.759, -56.358, 119.665, -81.896, 60.19, 154.058]
  Print: /'Cut out part'
  Set speed (100.0 mm/s)
  MoveL 875 to (-197.68, 45.77, 34.52) mm, rotated rx -180 ry 0 rz -11.91 deg; joints [12.927, -47.759, 117.761, -88.818, 90.006, 159.137]
  MoveL 876 to (-197.68, 45.77, 3.11) mm, rotated rx 180 ry 0 rz -11.91 deg; joints [12.937, -45.836, 117.514, -88.809, 89.974, 160.813]
  Set speed (25.4 mm/s)
  MoveL 877 to (-197.68, 45.77, -0.84) mm, rotated rx 180 ry 0 rz -11.91 deg; joints [12.938, -45.592, 117.477, -88.808, 89.97, 161.02]
  MoveL 878 to (-197.57, 46.4, -1.47) mm, rotated rx -180 ry 0 rz -11.91 deg; joints [12.936, -45.531, 117.418, -88.81, 89.97, 161.022]
  Set speed (38.1 mm/s)
  MoveL 879 to (-197.51, 46.74, -1.47) mm, rotated rx -180 ry 0 rz -11.91 deg; joints [12.936, -45.519, 117.388, -88.81, 89.97, 161.004]
  MoveL 880 to (-196.6, 47.2, -1.47) mm, rotated rx -180 ry 0 rz -11.91 deg; joints [12.969, -45.497, 117.333, -88.779, 89.981, 160.971]
  Set speed (76.2 mm/s)
  MoveL 881 to (-196.42, 47.11, -1.47) mm, rotated rx 180 ry 0 rz -11.91 deg; joints [12.978, -45.499, 117.337, -88.771, 89.984, 160.974]
  MoveL 882 to (-196.18, 47.01, -1.48) mm, rotated rx -180 ry 0 rz -11.91 deg; joints [12.989, -45.501, 117.341, -88.76, 89.987, 160.976]
  MoveL 883 to (-195.93, 46.94, -1.48) mm, rotated rx 180 ry 0 rz -11.91 deg; joints [12.999, -45.501, 117.342, -88.75, 89.99, 160.977]
  MoveL 884 to (-195.69, 46.88, -1.48) mm, rotated rx 180 ry 0 rz -11.91 deg; joints [13.01, -45.501, 117.342, -88.74, 89.994, 160.977]
  MoveL 885 to (-195.45, 46.84, -1.47) mm, rotated rx 180 ry 0 rz -11.91 deg; joints [13.02, -45.501, 117.341, -88.73, 89.997, 160.976]
  MoveL 886 to (-195.21, 46.83, -1.48) mm, rotated rx -180 ry 0 rz -11.91 deg; joints [13.031, -45.5, 117.338, -88.72, 90, 160.974]
  MoveL 887 to (-194.97, 46.83, -1.48) mm, rotated rx -180 ry 0 rz -11.91 deg; joints [13.041, -45.498, 117.333, -88.711, 90.003, 160.971]
  MoveL 888 to (213.41, 46.82, -1.48) mm, rotated rx 180 ry 0 rz -11.91 deg; joints [28.561, -40.236, 104.445, -74.672, 96.84, 154.321]
  MoveL 889 to (213.89, 46.83, -1.48) mm, rotated rx 180 ry 0 rz -11.91 deg; joints [28.577, -40.227, 104.423, -74.659, 96.85, 154.311]
  MoveL 890 to (214.13, 46.85, -1.48) mm, rotated rx 180 ry 0 rz -11.91 deg; joints [28.585, -40.221, 104.411, -74.652, 96.855, 154.305]
  MoveL 891 to (214.37, 46.9, -1.48) mm, rotated rx -180 ry 0 rz -11.91 deg; joints [28.593, -40.215, 104.397, -74.647, 96.86, 154.298]
  MoveL 892 to (214.63, 46.96, -1.47) mm, rotated rx -180 ry 0 rz -11.91 deg; joints [28.6, -40.208, 104.38, -74.641, 96.866, 154.289]
  MoveL 893 to (214.88, 47.05, -1.47) mm, rotated rx 180 ry 0 rz -11.91 deg; joints [28.607, -40.2, 104.361, -74.636, 96.872, 154.28]
  MoveL 894 to (215.01, 47.11, -1.48) mm, rotated rx -180 ry 0 rz -11.91 deg; joints [28.61, -40.196, 104.351, -74.634, 96.875, 154.275]
  MoveL 895 to (215.14, 47.17, -1.47) mm, rotated rx 180 ry 0 rz -11.91 deg; joints [28.613, -40.191, 104.341, -74.631, 96.878, 154.269]
  MoveL 896 to (215.26, 47.23, -1.47) mm, rotated rx -180 ry 0 rz -11.91 deg; joints [28.616, -40.186, 104.33, -74.629, 96.881, 154.263]
  MoveL 897 to (215.39, 47.31, -1.48) mm, rotated rx -180 ry 0 rz -11.91 deg; joints [28.619, -40.181, 104.318, -74.627, 96.884, 154.257]
  MoveL 898 to (215.62, 47.47, -1.48) mm, rotated rx -180 ry 0 rz -11.91 deg; joints [28.624, -40.171, 104.295, -74.625, 96.889, 154.245]
  MoveL 899 to (215.84, 47.66, -1.47) mm, rotated rx -180 ry 0 rz -11.91 deg; joints [28.628, -40.16, 104.27, -74.622, 96.895, 154.232]
  MoveL 900 to (215.98, 47.78, -1.48) mm, rotated rx 180 ry 0 rz -11.91 deg; joints [28.63, -40.153, 104.253, -74.622, 96.898, 154.223]
  MoveL 901 to (216.1, 47.91, -1.47) mm, rotated rx -180 ry 0 rz -11.91 deg; joints [28.632, -40.146, 104.238, -74.621, 96.901, 154.215]
  MoveL 902 to (216.2, 48.04, -1.47) mm, rotated rx -180 ry 0 rz -11.91 deg; joints [28.633, -40.14, 104.222, -74.621, 96.904, 154.206]
  MoveL 903 to (216.3, 48.17, -1.47) mm, rotated rx -180 ry 0 rz -11.91 deg; joints [28.634, -40.133, 104.208, -74.621, 96.906, 154.198]
  MoveL 904 to (216.39, 48.31, -1.47) mm, rotated rx -180 ry 0 rz -11.91 deg; joints [28.635, -40.127, 104.193, -74.622, 96.909, 154.19]
  MoveL 905 to (216.47, 48.44, -1.47) mm, rotated rx -180 ry 0 rz -11.91 deg; joints [28.635, -40.121, 104.178, -74.622, 96.911, 154.182]
  MoveL 906 to (216.54, 48.57, -1.48) mm, rotated rx -180 ry 0 rz -11.91 deg; joints [28.635, -40.115, 104.164, -74.623, 96.913, 154.175]
  MoveL 907 to (216.6, 48.71, -1.48) mm, rotated rx -180 ry 0 rz -11.91 deg; joints [28.634, -40.109, 104.151, -74.625, 96.915, 154.167]
  MoveL 908 to (216.66, 48.84, -1.48) mm, rotated rx 180 ry 0 rz -11.91 deg; joints [28.634, -40.103, 104.137, -74.626, 96.917, 154.16]
  MoveL 909 to (216.71, 48.97, -1.48) mm, rotated rx -180 ry 0 rz -11.91 deg; joints [28.633, -40.097, 104.124, -74.628, 96.918, 154.153]
  MoveL 910 to (216.75, 49.11, -1.48) mm, rotated rx -180 ry 0 rz -11.91 deg; joints [28.632, -40.091, 104.111, -74.629, 96.92, 154.145]
  MoveL 911 to (216.79, 49.24, -1.47) mm, rotated rx -180 ry 0 rz -11.91 deg; joints [28.631, -40.086, 104.099, -74.631, 96.921, 154.139]
  MoveL 912 to (216.84, 49.48, -1.48) mm, rotated rx -180 ry 0 rz -11.91 deg; joints [28.628, -40.076, 104.077, -74.635, 96.923, 154.126]
  MoveL 913 to (216.87, 49.73, -1.47) mm, rotated rx -180 ry 0 rz -11.91 deg; joints [28.624, -40.067, 104.056, -74.64, 96.925, 154.114]
  MoveL 914 to (216.88, 49.97, -1.48) mm, rotated rx 180 ry 0 rz -11.91 deg; joints [28.62, -40.058, 104.036, -74.645, 96.926, 154.103]
  MoveL 915 to (216.87, 50.21, -1.47) mm, rotated rx 180 ry 0 rz -11.91 deg; joints [28.616, -40.05, 104.017, -74.65, 96.927, 154.092]
  MoveL 916 to (216.85, 50.45, -1.48) mm, rotated rx 180 ry 0 rz -11.91 deg; joints [28.61, -40.042, 103.998, -74.657, 96.928, 154.081]
  MoveL 917 to (216.8, 50.69, -1.48) mm, rotated rx 180 ry 0 rz -11.91 deg; joints [28.604, -40.034, 103.98, -74.663, 96.928, 154.071]
  MoveL 918 to (216.74, 50.93, -1.47) mm, rotated rx -180 ry 0 rz -11.91 deg; joints [28.598, -40.026, 103.964, -74.67, 96.927, 154.061]
  MoveL 919 to (216.65, 51.17, -1.48) mm, rotated rx 180 ry 0 rz -11.91 deg; joints [28.591, -40.019, 103.948, -74.678, 96.927, 154.052]
  MoveL 920 to (216.58, 51.34, -1.48) mm, rotated rx 180 ry 0 rz -11.91 deg; joints [28.585, -40.015, 103.938, -74.684, 96.926, 154.045]
  MoveL 921 to (216.5, 51.5, -1.48) mm, rotated rx -180 ry 0 rz -11.91 deg; joints [28.579, -40.011, 103.928, -74.689, 96.925, 154.04]
  MoveL 922 to (216.41, 51.67, -1.48) mm, rotated rx -180 ry 0 rz -11.91 deg; joints [28.573, -40.006, 103.919, -74.696, 96.923, 154.034]
  MoveL 923 to (216.3, 51.83, -1.47) mm, rotated rx -180 ry 0 rz -11.91 deg; joints [28.567, -40.003, 103.91, -74.702, 96.922, 154.029]
  MoveL 924 to (216.2, 51.96, -1.47) mm, rotated rx 180 ry 0 rz -11.91 deg; joints [28.561, -40, 103.904, -74.708, 96.92, 154.024]
  MoveL 925 to (216.09, 52.1, -1.47) mm, rotated rx 180 ry 0 rz -11.91 deg; joints [28.554, -39.997, 103.898, -74.714, 96.919, 154.02]
  MoveL 926 to (215.96, 52.23, -1.47) mm, rotated rx -180 ry 0 rz -11.91 deg; joints [28.548, -39.995, 103.892, -74.721, 96.916, 154.017]
  MoveL 927 to (215.82, 52.37, -1.47) mm, rotated rx -180 ry 0 rz -11.91 deg; joints [28.54, -39.992, 103.888, -74.728, 96.914, 154.013]
  MoveL 928 to (215.58, 52.56, -1.47) mm, rotated rx -180 ry 0 rz -11.91 deg; joints [28.529, -39.99, 103.882, -74.739, 96.91, 154.009]
  MoveL 929 to (215.34, 52.72, -1.48) mm, rotated rx 180 ry 0 rz -11.91 deg; joints [28.518, -39.989, 103.88, -74.749, 96.905, 154.007]
  MoveL 930 to (215.09, 52.85, -1.47) mm, rotated rx -180 ry 0 rz -11.91 deg; joints [28.507, -39.989, 103.88, -74.758, 96.901, 154.006]
  MoveL 931 to (214.85, 52.96, -1.47) mm, rotated rx -180 ry 0 rz -11.91 deg; joints [28.497, -39.989, 103.882, -74.767, 96.896, 154.006]
  MoveL 932 to (214.61, 53.04, -1.48) mm, rotated rx -180 ry 0 rz -11.91 deg; joints [28.487, -39.991, 103.886, -74.776, 96.892, 154.007]
  MoveL 933 to (214.37, 53.1, -1.47) mm, rotated rx -180 ry 0 rz -11.91 deg; joints [28.478, -39.993, 103.892, -74.784, 96.887, 154.009]
  MoveL 934 to (214.36, 53.11, -1.48) mm, rotated rx -180 ry 0 rz -11.91 deg; joints [28.478, -39.994, 103.892, -74.785, 96.886, 154.01]
  MoveL 935 to (214.12, 53.15, -1.48) mm, rotated rx -180 ry 0 rz -11.91 deg; joints [28.469, -39.997, 103.899, -74.792, 96.882, 154.013]
  MoveL 936 to (213.88, 53.17, -1.47) mm, rotated rx -180 ry 0 rz -11.91 deg; joints [28.46, -40, 103.908, -74.799, 96.877, 154.017]
  MoveL 937 to (213.4, 53.17, -1.47) mm, rotated rx -180 ry 0 rz -11.91 deg; joints [28.444, -40.009, 103.929, -74.813, 96.867, 154.026]
  MoveL 938 to (-195.12, 53.17, -1.47) mm, rotated rx -180 ry 0 rz -11.91 deg; joints [12.973, -45.286, 116.815, -88.775, 89.989, 160.665]
  MoveL 939 to (-195.28, 53.17, -1.48) mm, rotated rx -180 ry 0 rz -11.91 deg; joints [12.967, -45.287, 116.819, -88.781, 89.987, 160.667]
  MoveL 940 to (-195.43, 53.16, -1.48) mm, rotated rx -180 ry 0 rz -11.91 deg; joints [12.96, -45.289, 116.823, -88.787, 89.985, 160.67]
  MoveL 941 to (-195.59, 53.14, -1.47) mm, rotated rx -180 ry 0 rz -11.91 deg; joints [12.954, -45.29, 116.828, -88.793, 89.982, 160.673]
  MoveL 942 to (-195.75, 53.11, -1.47) mm, rotated rx -180 ry 0 rz -11.91 deg; joints [12.948, -45.293, 116.833, -88.799, 89.98, 160.676]
  MoveL 943 to (-195.92, 53.07, -1.48) mm, rotated rx -180 ry 0 rz -11.91 deg; joints [12.941, -45.295, 116.839, -88.805, 89.978, 160.68]
  MoveL 944 to (-196.08, 53.02, -1.47) mm, rotated rx -180 ry 0 rz -11.91 deg; joints [12.935, -45.298, 116.847, -88.811, 89.976, 160.684]
  MoveL 945 to (-196.25, 52.96, -1.47) mm, rotated rx 180 ry 0 rz -11.91 deg; joints [12.928, -45.301, 116.855, -88.817, 89.974, 160.689]
  MoveL 946 to (-196.42, 52.89, -1.48) mm, rotated rx -180 ry 0 rz -11.91 deg; joints [12.922, -45.305, 116.864, -88.823, 89.972, 160.694]
  MoveL 947 to (-196.56, 52.82, -1.48) mm, rotated rx -180 ry 0 rz -11.91 deg; joints [12.917, -45.308, 116.872, -88.828, 89.97, 160.699]
  MoveL 948 to (-196.7, 52.74, -1.47) mm, rotated rx -180 ry 0 rz -11.91 deg; joints [12.912, -45.312, 116.881, -88.833, 89.969, 160.704]
  MoveL 949 to (-196.84, 52.66, -1.48) mm, rotated rx -180 ry 0 rz -11.91 deg; joints [12.907, -45.316, 116.891, -88.838, 89.967, 160.71]
  MoveL 950 to (-196.98, 52.56, -1.48) mm, rotated rx -180 ry 0 rz -11.91 deg; joints [12.902, -45.32, 116.901, -88.842, 89.965, 160.716]
  MoveL 951 to (-197.12, 52.45, -1.47) mm, rotated rx -180 ry 0 rz -11.91 deg; joints [12.897, -45.325, 116.913, -88.847, 89.963, 160.723]
  MoveL 952 to (-197.26, 52.33, -1.48) mm, rotated rx -180 ry 0 rz -11.91 deg; joints [12.892, -45.33, 116.926, -88.851, 89.962, 160.731]
  MoveL 953 to (-197.41, 52.18, -1.48) mm, rotated rx 180 ry 0 rz -11.91 deg; joints [12.888, -45.336, 116.941, -88.856, 89.96, 160.739]
  MoveL 954 to (-197.54, 52.03, -1.48) mm, rotated rx -180 ry 0 rz -11.91 deg; joints [12.884, -45.342, 116.955, -88.86, 89.959, 160.748]
  MoveL 955 to (-197.7, 51.82, -1.48) mm, rotated rx -180 ry 0 rz -11.91 deg; joints [12.879, -45.35, 116.976, -88.864, 89.957, 160.76]
  MoveL 956 to (-197.84, 51.6, -1.47) mm, rotated rx -180 ry 0 rz -11.91 deg; joints [12.875, -45.359, 116.996, -88.868, 89.956, 160.772]
  MoveL 957 to (-197.95, 51.39, -1.47) mm, rotated rx -180 ry 0 rz -11.91 deg; joints [12.872, -45.367, 117.016, -88.87, 89.955, 160.784]
  MoveL 958 to (-198.05, 51.18, -1.48) mm, rotated rx -180 ry 0 rz -11.91 deg; joints [12.871, -45.374, 117.035, -88.872, 89.954, 160.795]
  MoveL 959 to (-198.13, 50.93, -1.48) mm, rotated rx 180 ry 0 rz -11.91 deg; joints [12.869, -45.383, 117.056, -88.873, 89.953, 160.808]
  MoveL 960 to (-198.2, 50.69, -1.47) mm, rotated rx -180 ry 0 rz -11.91 deg; joints [12.869, -45.392, 117.077, -88.874, 89.953, 160.82]
  MoveL 961 to (-198.24, 50.45, -1.47) mm, rotated rx 180 ry 0 rz -11.91 deg; joints [12.869, -45.4, 117.098, -88.873, 89.953, 160.833]
  MoveL 962 to (-198.27, 50.21, -1.47) mm, rotated rx -180 ry 0 rz -11.91 deg; joints [12.871, -45.409, 117.118, -88.872, 89.953, 160.845]
  MoveL 963 to (-198.27, 49.97, -1.48) mm, rotated rx -180 ry 0 rz -11.91 deg; joints [12.873, -45.417, 117.138, -88.87, 89.953, 160.856]
  MoveL 964 to (-198.26, 49.73, -1.48) mm, rotated rx 180 ry 0 rz -11.91 deg; joints [12.876, -45.425, 117.158, -88.867, 89.954, 160.868]
  MoveL 965 to (-198.23, 49.48, -1.47) mm, rotated rx 180 ry 0 rz -11.91 deg; joints [12.879, -45.433, 117.177, -88.864, 89.955, 160.879]
  MoveL 966 to (-198.18, 49.24, -1.48) mm, rotated rx -180 ry 0 rz -11.91 deg; joints [12.884, -45.44, 117.196, -88.86, 89.956, 160.891]
  MoveL 967 to (-198.11, 49, -1.48) mm, rotated rx -180 ry 0 rz -11.91 deg; joints [12.889, -45.448, 117.215, -88.855, 89.957, 160.901]
  MoveL 968 to (-198.02, 48.76, -1.48) mm, rotated rx 180 ry 0 rz -11.91 deg; joints [12.895, -45.455, 117.233, -88.849, 89.959, 160.912]
  MoveL 969 to (-197.91, 48.52, -1.48) mm, rotated rx -180 ry 0 rz -11.91 deg; joints [12.902, -45.463, 117.25, -88.842, 89.961, 160.923]
  MoveL 970 to (-197.76, 48.28, -1.48) mm, rotated rx 180 ry 0 rz -11.91 deg; joints [12.91, -45.47, 117.267, -88.835, 89.963, 160.933]
  MoveL 971 to (-197.66, 48.13, -1.48) mm, rotated rx 180 ry 0 rz -11.91 deg; joints [12.916, -45.474, 117.278, -88.829, 89.965, 160.939]
  MoveL 972 to (-197.55, 47.98, -1.47) mm, rotated rx 180 ry 0 rz -11.91 deg; joints [12.922, -45.478, 117.287, -88.823, 89.967, 160.944]
  MoveL 973 to (-197.42, 47.84, -1.48) mm, rotated rx 180 ry 0 rz -11.91 deg; joints [12.929, -45.482, 117.297, -88.817, 89.969, 160.95]
  MoveL 974 to (-197.27, 47.69, -1.47) mm, rotated rx -180 ry 0 rz -11.91 deg; joints [12.936, -45.486, 117.306, -88.81, 89.971, 160.956]
  MoveL 975 to (-197.03, 47.48, -1.47) mm, rotated rx -180 ry 0 rz -11.91 deg; joints [12.948, -45.491, 117.319, -88.798, 89.975, 160.963]
  MoveL 976 to (-196.78, 47.31, -1.47) mm, rotated rx -180 ry 0 rz -11.91 deg; joints [12.96, -45.495, 117.328, -88.787, 89.978, 160.968]
  MoveL 977 to (-196.6, 47.2, -1.47) mm, rotated rx -180 ry 0 rz -11.91 deg; joints [12.969, -45.497, 117.333, -88.779, 89.981, 160.971]
  Set speed (38.1 mm/s)
  MoveL 978 to (-197.17, 46.07, -1.47) mm, rotated rx -180 ry 0 rz -11.91 deg; joints [12.956, -45.539, 117.437, -88.791, 89.976, 161.033]
  MoveL 979 to (-197.73, 46.35, -1.47) mm, rotated rx -180 ry 0 rz -11.91 deg; joints [12.93, -45.534, 117.425, -88.816, 89.968, 161.026]
  Set speed (25.4 mm/s)
  MoveL 980 to (-197.73, 46.35, -3.84) mm, rotated rx 180 ry 0 rz -11.91 deg; joints [12.931, -45.388, 117.402, -88.815, 89.965, 161.149]
  MoveL 981 to (-197.45, 46.92, -4.47) mm, rotated rx 180 ry 0 rz -11.91 deg; joints [12.937, -45.328, 117.344, -88.809, 89.967, 161.151]
  Set speed (38.1 mm/s)
  MoveL 982 to (-196.6, 47.2, -4.47) mm, rotated rx -180 ry 0 rz -11.91 deg; joints [12.97, -45.312, 117.304, -88.778, 89.978, 161.128]
  Set speed (76.2 mm/s)
  MoveL 983 to (-196.42, 47.11, -4.47) mm, rotated rx -180 ry 0 rz -11.91 deg; joints [12.978, -45.314, 117.308, -88.77, 89.98, 161.13]
  MoveL 984 to (-196.18, 47.01, -4.48) mm, rotated rx 180 ry 0 rz -11.91 deg; joints [12.989, -45.315, 117.312, -88.759, 89.984, 161.132]
  MoveL 985 to (-195.93, 46.94, -4.48) mm, rotated rx 180 ry 0 rz -11.91 deg; joints [13, -45.316, 117.313, -88.749, 89.987, 161.133]
  MoveL 986 to (-195.69, 46.88, -4.48) mm, rotated rx -180 ry 0 rz -11.91 deg; joints [13.011, -45.316, 117.313, -88.739, 89.99, 161.133]
  MoveL 987 to (-195.45, 46.84, -4.48) mm, rotated rx -180 ry 0 rz -11.91 deg; joints [13.021, -45.316, 117.312, -88.729, 89.994, 161.132]
  MoveL 988 to (-195.21, 46.83, -4.47) mm, rotated rx 180 ry 0 rz -11.91 deg; joints [13.031, -45.314, 117.309, -88.719, 89.997, 161.13]
  MoveL 989 to (-194.97, 46.83, -4.48) mm, rotated rx 180 ry 0 rz -11.91 deg; joints [13.042, -45.313, 117.304, -88.71, 90, 161.127]
  MoveL 990 to (213.41, 46.82, -4.47) mm, rotated rx -180 ry 0 rz -11.91 deg; joints [28.562, -40.073, 104.417, -74.655, 96.805, 154.453]
  MoveL 991 to (213.89, 46.83, -4.47) mm, rotated rx 180 ry 0 rz -11.91 deg; joints [28.579, -40.064, 104.396, -74.642, 96.815, 154.442]
  MoveL 992 to (214.13, 46.85, -4.47) mm, rotated rx -180 ry 0 rz -11.91 deg; joints [28.586, -40.058, 104.383, -74.636, 96.82, 154.436]
  MoveL 993 to (214.37, 46.9, -4.47) mm, rotated rx 180 ry 0 rz -11.91 deg; joints [28.594, -40.052, 104.369, -74.63, 96.825, 154.429]
  MoveL 994 to (214.63, 46.96, -4.47) mm, rotated rx 180 ry 0 rz -11.91 deg; joints [28.601, -40.045, 104.352, -74.624, 96.831, 154.421]
  MoveL 995 to (214.88, 47.05, -4.47) mm, rotated rx 180 ry 0 rz -11.91 deg; joints [28.608, -40.037, 104.334, -74.619, 96.836, 154.411]
  MoveL 996 to (215.01, 47.11, -4.47) mm, rotated rx -180 ry 0 rz -11.91 deg; joints [28.611, -40.033, 104.324, -74.617, 96.839, 154.406]
  MoveL 997 to (215.14, 47.17, -4.47) mm, rotated rx -180 ry 0 rz -11.91 deg; joints [28.615, -40.028, 104.313, -74.614, 96.842, 154.401]
  MoveL 998 to (215.26, 47.23, -4.48) mm, rotated rx -180 ry 0 rz -11.91 deg; joints [28.618, -40.023, 104.302, -74.612, 96.845, 154.395]
  MoveL 999 to (215.39, 47.31, -4.47) mm, rotated rx -180 ry 0 rz -11.91 deg; joints [28.621, -40.018, 104.29, -74.611, 96.848, 154.389]
  MoveL 1000 to (215.62, 47.47, -4.48) mm, rotated rx 180 ry 0 rz -11.91 deg; joints [28.625, -40.009, 104.267, -74.608, 96.854, 154.377]
  MoveL 1001 to (215.84, 47.66, -4.47) mm, rotated rx -180 ry 0 rz -11.91 deg; joints [28.63, -39.998, 104.242, -74.606, 96.859, 154.363]
  MoveL 1002 to (215.98, 47.78, -4.47) mm, rotated rx -180 ry 0 rz -11.91 deg; joints [28.632, -39.99, 104.226, -74.605, 96.863, 154.354]
  MoveL 1003 to (216.1, 47.91, -4.48) mm, rotated rx 180 ry 0 rz -11.91 deg; joints [28.633, -39.984, 104.21, -74.604, 96.866, 154.346]
  MoveL 1004 to (216.2, 48.04, -4.48) mm, rotated rx -180 ry 0 rz -11.91 deg; joints [28.634, -39.977, 104.195, -74.604, 96.868, 154.338]
  MoveL 1005 to (216.3, 48.17, -4.48) mm, rotated rx -180 ry 0 rz -11.91 deg; joints [28.635, -39.971, 104.18, -74.604, 96.871, 154.33]
  MoveL 1006 to (216.39, 48.31, -4.48) mm, rotated rx -180 ry 0 rz -11.91 deg; joints [28.636, -39.964, 104.165, -74.605, 96.873, 154.322]
  MoveL 1007 to (216.47, 48.44, -4.48) mm, rotated rx -180 ry 0 rz -11.91 deg; joints [28.636, -39.958, 104.151, -74.606, 96.876, 154.314]
  MoveL 1008 to (216.54, 48.57, -4.47) mm, rotated rx -180 ry 0 rz -11.91 deg; joints [28.636, -39.952, 104.137, -74.607, 96.878, 154.306]
  MoveL 1009 to (216.6, 48.71, -4.47) mm, rotated rx -180 ry 0 rz -11.91 deg; joints [28.636, -39.946, 104.123, -74.608, 96.88, 154.299]
  MoveL 1010 to (216.66, 48.84, -4.48) mm, rotated rx 180 ry 0 rz -11.91 deg; joints [28.635, -39.94, 104.11, -74.609, 96.881, 154.291]
  MoveL 1011 to (216.71, 48.97, -4.48) mm, rotated rx 180 ry 0 rz -11.91 deg; joints [28.634, -39.934, 104.097, -74.611, 96.883, 154.284]
  MoveL 1012 to (216.75, 49.11, -4.47) mm, rotated rx -180 ry 0 rz -11.91 deg; joints [28.633, -39.929, 104.084, -74.613, 96.885, 154.277]
  MoveL 1013 to (216.79, 49.24, -4.47) mm, rotated rx -180 ry 0 rz -11.91 deg; joints [28.632, -39.923, 104.071, -74.614, 96.886, 154.27]
  MoveL 1014 to (216.84, 49.48, -4.48) mm, rotated rx -180 ry 0 rz -11.91 deg; joints [28.629, -39.914, 104.049, -74.618, 96.888, 154.257]
  MoveL 1015 to (216.87, 49.73, -4.48) mm, rotated rx -180 ry 0 rz -11.91 deg; joints [28.626, -39.905, 104.029, -74.623, 96.89, 154.246]
  MoveL 1016 to (216.88, 49.97, -4.48) mm, rotated rx 180 ry 0 rz -11.91 deg; joints [28.622, -39.896, 104.008, -74.628, 96.891, 154.234]
  MoveL 1017 to (216.87, 50.21, -4.48) mm, rotated rx -180 ry 0 rz -11.91 deg; joints [28.617, -39.887, 103.989, -74.634, 96.892, 154.223]
  MoveL 1018 to (216.85, 50.45, -4.47) mm, rotated rx -180 ry 0 rz -11.91 deg; joints [28.612, -39.879, 103.97, -74.64, 96.892, 154.212]
  MoveL 1019 to (216.8, 50.69, -4.47) mm, rotated rx 180 ry 0 rz -11.91 deg; joints [28.606, -39.871, 103.953, -74.646, 96.892, 154.202]
  MoveL 1020 to (216.74, 50.93, -4.47) mm, rotated rx 180 ry 0 rz -11.91 deg; joints [28.599, -39.864, 103.936, -74.653, 96.892, 154.192]
  MoveL 1021 to (216.65, 51.18, -4.48) mm, rotated rx 180 ry 0 rz -11.91 deg; joints [28.592, -39.857, 103.92, -74.661, 96.891, 154.183]
  MoveL 1022 to (216.58, 51.34, -4.48) mm, rotated rx -180 ry 0 rz -11.91 deg; joints [28.586, -39.852, 103.91, -74.667, 96.891, 154.177]
  MoveL 1023 to (216.5, 51.5, -4.48) mm, rotated rx -180 ry 0 rz -11.91 deg; joints [28.581, -39.848, 103.9, -74.673, 96.89, 154.171]
  MoveL 1024 to (216.41, 51.67, -4.47) mm, rotated rx 180 ry 0 rz -11.91 deg; joints [28.574, -39.844, 103.891, -74.679, 96.888, 154.165]
  MoveL 1025 to (216.3, 51.83, -4.47) mm, rotated rx 180 ry 0 rz -11.91 deg; joints [28.568, -39.84, 103.883, -74.685, 96.887, 154.16]
  MoveL 1026 to (216.2, 51.96, -4.47) mm, rotated rx -180 ry 0 rz -11.91 deg; joints [28.562, -39.837, 103.876, -74.691, 96.885, 154.155]
  MoveL 1027 to (216.09, 52.1, -4.48) mm, rotated rx 180 ry 0 rz -11.91 deg; joints [28.556, -39.835, 103.87, -74.697, 96.884, 154.151]
  MoveL 1028 to (215.96, 52.23, -4.48) mm, rotated rx -180 ry 0 rz -11.91 deg; joints [28.549, -39.832, 103.865, -74.704, 96.881, 154.148]
  MoveL 1029 to (215.82, 52.37, -4.48) mm, rotated rx -180 ry 0 rz -11.91 deg; joints [28.542, -39.83, 103.86, -74.711, 96.879, 154.144]
  MoveL 1030 to (215.58, 52.56, -4.48) mm, rotated rx 180 ry 0 rz -11.91 deg; joints [28.53, -39.828, 103.855, -74.722, 96.875, 154.14]
  MoveL 1031 to (215.34, 52.72, -4.48) mm, rotated rx 180 ry 0 rz -11.91 deg; joints [28.519, -39.826, 103.852, -74.732, 96.87, 154.138]
  MoveL 1032 to (215.09, 52.85, -4.48) mm, rotated rx -180 ry 0 rz -11.91 deg; joints [28.508, -39.826, 103.852, -74.742, 96.866, 154.137]
  MoveL 1033 to (214.85, 52.96, -4.47) mm, rotated rx 180 ry 0 rz -11.91 deg; joints [28.498, -39.827, 103.855, -74.751, 96.861, 154.137]
  MoveL 1034 to (214.61, 53.04, -4.48) mm, rotated rx -180 ry 0 rz -11.91 deg; joints [28.489, -39.829, 103.858, -74.759, 96.857, 154.138]
  MoveL 1035 to (214.37, 53.1, -4.47) mm, rotated rx -180 ry 0 rz -11.91 deg; joints [28.479, -39.831, 103.864, -74.767, 96.852, 154.14]
  MoveL 1036 to (214.36, 53.11, -4.48) mm, rotated rx 180 ry 0 rz -11.91 deg; joints [28.479, -39.831, 103.865, -74.768, 96.852, 154.141]
  MoveL 1037 to (214.12, 53.15, -4.47) mm, rotated rx -180 ry 0 rz -11.91 deg; joints [28.47, -39.834, 103.872, -74.775, 96.847, 154.144]
  MoveL 1038 to (213.88, 53.17, -4.48) mm, rotated rx 180 ry 0 rz -11.91 deg; joints [28.462, -39.838, 103.881, -74.782, 96.842, 154.148]
  MoveL 1039 to (213.4, 53.17, -4.47) mm, rotated rx 180 ry 0 rz -11.91 deg; joints [28.445, -39.847, 103.901, -74.796, 96.832, 154.157]
  MoveL 1040 to (-195.12, 53.17, -4.48) mm, rotated rx -180 ry 0 rz -11.91 deg; joints [12.974, -45.101, 116.786, -88.774, 89.986, 160.821]
  MoveL 1041 to (-195.28, 53.17, -4.47) mm, rotated rx 180 ry 0 rz -11.91 deg; joints [12.967, -45.103, 116.79, -88.78, 89.984, 160.823]
  MoveL 1042 to (-195.43, 53.16, -4.48) mm, rotated rx -180 ry 0 rz -11.91 deg; joints [12.961, -45.104, 116.794, -88.786, 89.982, 160.825]
  MoveL 1043 to (-195.59, 53.14, -4.48) mm, rotated rx -180 ry 0 rz -11.91 deg; joints [12.955, -45.106, 116.799, -88.792, 89.98, 160.828]
  MoveL 1044 to (-195.75, 53.11, -4.47) mm, rotated rx -180 ry 0 rz -11.91 deg; joints [12.948, -45.108, 116.804, -88.798, 89.977, 160.831]
  MoveL 1045 to (-195.92, 53.07, -4.48) mm, rotated rx -180 ry 0 rz -11.91 deg; joints [12.942, -45.111, 116.81, -88.804, 89.975, 160.835]
  MoveL 1046 to (-196.08, 53.02, -4.48) mm, rotated rx -180 ry 0 rz -11.91 deg; joints [12.935, -45.114, 116.818, -88.811, 89.973, 160.839]
  MoveL 1047 to (-196.25, 52.96, -4.48) mm, rotated rx 180 ry 0 rz -11.91 deg; joints [12.929, -45.117, 116.826, -88.817, 89.971, 160.844]
  MoveL 1048 to (-196.42, 52.89, -4.48) mm, rotated rx -180 ry 0 rz -11.91 deg; joints [12.923, -45.121, 116.835, -88.822, 89.969, 160.849]
  MoveL 1049 to (-196.56, 52.82, -4.47) mm, rotated rx 180 ry 0 rz -11.91 deg; joints [12.918, -45.124, 116.843, -88.827, 89.967, 160.854]
  MoveL 1050 to (-196.7, 52.74, -4.48) mm, rotated rx 180 ry 0 rz -11.91 deg; joints [12.913, -45.127, 116.852, -88.832, 89.966, 160.859]
  MoveL 1051 to (-196.84, 52.66, -4.48) mm, rotated rx 180 ry 0 rz -11.91 deg; joints [12.908, -45.131, 116.862, -88.837, 89.964, 160.865]
  MoveL 1052 to (-196.98, 52.56, -4.48) mm, rotated rx -180 ry 0 rz -11.91 deg; joints [12.903, -45.136, 116.872, -88.842, 89.962, 160.872]
  MoveL 1053 to (-197.12, 52.45, -4.48) mm, rotated rx -180 ry 0 rz -11.91 deg; joints [12.898, -45.14, 116.884, -88.846, 89.961, 160.878]
  MoveL 1054 to (-197.26, 52.33, -4.48) mm, rotated rx -180 ry 0 rz -11.91 deg; joints [12.893, -45.145, 116.897, -88.851, 89.959, 160.886]
  MoveL 1055 to (-197.41, 52.18, -4.48) mm, rotated rx -180 ry 0 rz -11.91 deg; joints [12.889, -45.152, 116.912, -88.855, 89.957, 160.895]
  MoveL 1056 to (-197.54, 52.03, -4.47) mm, rotated rx -180 ry 0 rz -11.91 deg; joints [12.884, -45.157, 116.926, -88.859, 89.956, 160.904]
  MoveL 1057 to (-197.7, 51.82, -4.48) mm, rotated rx -180 ry 0 rz -11.91 deg; joints [12.88, -45.166, 116.947, -88.863, 89.954, 160.916]
  MoveL 1058 to (-197.84, 51.6, -4.48) mm, rotated rx -180 ry 0 rz -11.91 deg; joints [12.876, -45.174, 116.967, -88.867, 89.953, 160.928]
  MoveL 1059 to (-197.95, 51.39, -4.47) mm, rotated rx -180 ry 0 rz -11.91 deg; joints [12.873, -45.182, 116.987, -88.87, 89.952, 160.94]
  MoveL 1060 to (-198.05, 51.18, -4.48) mm, rotated rx -180 ry 0 rz -11.91 deg; joints [12.872, -45.19, 117.006, -88.871, 89.951, 160.951]
  MoveL 1061 to (-198.13, 50.93, -4.47) mm, rotated rx -180 ry 0 rz -11.91 deg; joints [12.87, -45.199, 117.027, -88.872, 89.95, 160.964]
  MoveL 1062 to (-198.2, 50.69, -4.48) mm, rotated rx -180 ry 0 rz -11.91 deg; joints [12.87, -45.207, 117.048, -88.873, 89.95, 160.976]
  MoveL 1063 to (-198.24, 50.45, -4.47) mm, rotated rx -180 ry 0 rz -11.91 deg; joints [12.87, -45.215, 117.069, -88.872, 89.95, 160.988]
  MoveL 1064 to (-198.27, 50.21, -4.47) mm, rotated rx -180 ry 0 rz -11.91 deg; joints [12.872, -45.224, 117.089, -88.871, 89.95, 161]
  MoveL 1065 to (-198.27, 49.97, -4.48) mm, rotated rx -180 ry 0 rz -11.91 deg; joints [12.874, -45.232, 117.109, -88.869, 89.95, 161.012]
  MoveL 1066 to (-198.26, 49.73, -4.47) mm, rotated rx -180 ry 0 rz -11.91 deg; joints [12.877, -45.24, 117.129, -88.867, 89.951, 161.024]
  MoveL 1067 to (-198.23, 49.48, -4.48) mm, rotated rx 180 ry 0 rz -11.91 deg; joints [12.88, -45.248, 117.148, -88.863, 89.952, 161.035]
  MoveL 1068 to (-198.18, 49.24, -4.48) mm, rotated rx 180 ry 0 rz -11.91 deg; joints [12.884, -45.255, 117.167, -88.859, 89.953, 161.046]
  MoveL 1069 to (-198.11, 49, -4.48) mm, rotated rx 180 ry 0 rz -11.91 deg; joints [12.89, -45.263, 117.185, -88.854, 89.954, 161.057]
  MoveL 1070 to (-198.02, 48.76, -4.47) mm, rotated rx 180 ry 0 rz -11.91 deg; joints [12.896, -45.27, 117.204, -88.848, 89.956, 161.068]
  MoveL 1071 to (-197.91, 48.52, -4.48) mm, rotated rx 180 ry 0 rz -11.91 deg; joints [12.903, -45.278, 117.221, -88.842, 89.958, 161.079]
  MoveL 1072 to (-197.76, 48.28, -4.48) mm, rotated rx 180 ry 0 rz -11.91 deg; joints [12.911, -45.285, 117.238, -88.834, 89.96, 161.089]
  MoveL 1073 to (-197.66, 48.13, -4.47) mm, rotated rx -180 ry 0 rz -11.91 deg; joints [12.917, -45.289, 117.248, -88.828, 89.962, 161.095]
  MoveL 1074 to (-197.55, 47.98, -4.47) mm, rotated rx -180 ry 0 rz -11.91 deg; joints [12.923, -45.293, 117.258, -88.823, 89.964, 161.101]
  MoveL 1075 to (-197.42, 47.84, -4.48) mm, rotated rx -180 ry 0 rz -11.91 deg; joints [12.93, -45.297, 117.268, -88.816, 89.966, 161.106]
  MoveL 1076 to (-197.27, 47.69, -4.47) mm, rotated rx 180 ry 0 rz -11.91 deg; joints [12.937, -45.301, 117.277, -88.809, 89.968, 161.112]
  MoveL 1077 to (-197.03, 47.48, -4.47) mm, rotated rx 180 ry 0 rz -11.91 deg; joints [12.949, -45.306, 117.29, -88.797, 89.972, 161.119]
  MoveL 1078 to (-196.78, 47.31, -4.47) mm, rotated rx -180 ry 0 rz -11.91 deg; joints [12.961, -45.31, 117.299, -88.786, 89.975, 161.125]
  MoveL 1079 to (-196.6, 47.2, -4.47) mm, rotated rx -180 ry 0 rz -11.91 deg; joints [12.97, -45.312, 117.304, -88.778, 89.978, 161.128]
  Set speed (38.1 mm/s)
  MoveL 1080 to (-197.17, 46.07, -4.48) mm, rotated rx -180 ry 0 rz -11.91 deg; joints [12.957, -45.354, 117.408, -88.79, 89.973, 161.189]
  MoveL 1081 to (-197.73, 46.35, -4.48) mm, rotated rx -180 ry 0 rz -11.91 deg; joints [12.931, -45.349, 117.396, -88.815, 89.965, 161.182]
  Set speed (25.4 mm/s)
  MoveL 1082 to (-197.73, 46.35, -6.84) mm, rotated rx -180 ry 0 rz -11.91 deg; joints [12.932, -45.202, 117.372, -88.814, 89.962, 161.305]
  MoveL 1083 to (-197.45, 46.92, -7.47) mm, rotated rx -180 ry 0 rz -11.91 deg; joints [12.938, -45.142, 117.314, -88.808, 89.964, 161.307]
  Set speed (38.1 mm/s)
  MoveL 1084 to (-196.6, 47.2, -7.47) mm, rotated rx -180 ry 0 rz -11.91 deg; joints [12.971, -45.126, 117.274, -88.777, 89.975, 161.283]
  Set speed (76.2 mm/s)
  MoveL 1085 to (-196.42, 47.11, -7.47) mm, rotated rx 180 ry 0 rz -11.91 deg; joints [12.979, -45.128, 117.278, -88.769, 89.977, 161.286]
  MoveL 1086 to (-196.18, 47.01, -7.47) mm, rotated rx -180 ry 0 rz -11.91 deg; joints [12.99, -45.13, 117.282, -88.758, 89.981, 161.288]
  MoveL 1087 to (-195.93, 46.94, -7.48) mm, rotated rx -180 ry 0 rz -11.91 deg; joints [13.001, -45.13, 117.284, -88.748, 89.984, 161.289]
  MoveL 1088 to (-195.69, 46.88, -7.48) mm, rotated rx -180 ry 0 rz -11.91 deg; joints [13.012, -45.131, 117.284, -88.738, 89.987, 161.289]
  MoveL 1089 to (-195.45, 46.84, -7.48) mm, rotated rx -180 ry 0 rz -11.91 deg; joints [13.022, -45.13, 117.282, -88.728, 89.99, 161.288]
  MoveL 1090 to (-195.21, 46.83, -7.48) mm, rotated rx 180 ry 0 rz -11.91 deg; joints [13.032, -45.129, 117.279, -88.718, 89.994, 161.286]
  MoveL 1091 to (-194.97, 46.82, -7.47) mm, rotated rx -180 ry 0 rz -11.91 deg; joints [13.042, -45.127, 117.274, -88.709, 89.997, 161.283]
  MoveL 1092 to (213.41, 46.82, -7.48) mm, rotated rx 180 ry 0 rz -11.91 deg; joints [28.564, -39.909, 104.389, -74.639, 96.769, 154.584]
  MoveL 1093 to (213.89, 46.83, -7.47) mm, rotated rx 180 ry 0 rz -11.91 deg; joints [28.58, -39.9, 104.367, -74.625, 96.78, 154.574]
  MoveL 1094 to (214.13, 46.85, -7.48) mm, rotated rx -180 ry 0 rz -11.91 deg; joints [28.588, -39.895, 104.355, -74.619, 96.785, 154.567]
  MoveL 1095 to (214.37, 46.9, -7.48) mm, rotated rx -180 ry 0 rz -11.91 deg; joints [28.595, -39.889, 104.341, -74.613, 96.79, 154.56]
  MoveL 1096 to (214.63, 46.96, -7.48) mm, rotated rx -180 ry 0 rz -11.91 deg; joints [28.602, -39.882, 104.324, -74.607, 96.795, 154.552]
  MoveL 1097 to (214.88, 47.05, -7.47) mm, rotated rx 180 ry 0 rz -11.91 deg; joints [28.609, -39.874, 104.305, -74.602, 96.801, 154.543]
  MoveL 1098 to (215.01, 47.11, -7.47) mm, rotated rx 180 ry 0 rz -11.91 deg; joints [28.613, -39.87, 104.295, -74.6, 96.804, 154.537]
  MoveL 1099 to (215.14, 47.17, -7.48) mm, rotated rx -180 ry 0 rz -11.91 deg; joints [28.616, -39.865, 104.285, -74.598, 96.807, 154.532]
  MoveL 1100 to (215.26, 47.23, -7.47) mm, rotated rx -180 ry 0 rz -11.91 deg; joints [28.619, -39.86, 104.274, -74.596, 96.81, 154.526]
  MoveL 1101 to (215.39, 47.31, -7.48) mm, rotated rx -180 ry 0 rz -11.91 deg; joints [28.622, -39.855, 104.262, -74.594, 96.813, 154.52]
  MoveL 1102 to (215.62, 47.47, -7.48) mm, rotated rx -180 ry 0 rz -11.91 deg; joints [28.627, -39.845, 104.239, -74.591, 96.818, 154.508]
  MoveL 1103 to (215.84, 47.66, -7.48) mm, rotated rx 180 ry 0 rz -11.91 deg; joints [28.631, -39.834, 104.214, -74.589, 96.824, 154.494]
  MoveL 1104 to (215.98, 47.78, -7.48) mm, rotated rx 180 ry 0 rz -11.91 deg; joints [28.633, -39.827, 104.197, -74.588, 96.827, 154.485]
  MoveL 1105 to (216.1, 47.91, -7.48) mm, rotated rx 180 ry 0 rz -11.91 deg; joints [28.635, -39.821, 104.182, -74.587, 96.83, 154.477]
  MoveL 1106 to (216.2, 48.04, -7.47) mm, rotated rx -180 ry 0 rz -11.91 deg; joints [28.636, -39.814, 104.166, -74.587, 96.833, 154.469]
  MoveL 1107 to (216.3, 48.17, -7.48) mm, rotated rx -180 ry 0 rz -11.91 deg; joints [28.637, -39.808, 104.152, -74.588, 96.836, 154.461]
  MoveL 1108 to (216.39, 48.31, -7.48) mm, rotated rx -180 ry 0 rz -11.91 deg; joints [28.637, -39.801, 104.137, -74.588, 96.838, 154.453]
  MoveL 1109 to (216.47, 48.44, -7.48) mm, rotated rx 180 ry 0 rz -11.91 deg; joints [28.637, -39.795, 104.122, -74.589, 96.84, 154.445]
  MoveL 1110 to (216.54, 48.57, -7.47) mm, rotated rx -180 ry 0 rz -11.91 deg; joints [28.637, -39.789, 104.108, -74.59, 96.843, 154.437]
  MoveL 1111 to (216.6, 48.71, -7.48) mm, rotated rx -180 ry 0 rz -11.91 deg; joints [28.637, -39.783, 104.095, -74.591, 96.845, 154.429]
  MoveL 1112 to (216.66, 48.84, -7.47) mm, rotated rx 180 ry 0 rz -11.91 deg; joints [28.636, -39.777, 104.081, -74.592, 96.846, 154.422]
  MoveL 1113 to (216.71, 48.97, -7.47) mm, rotated rx 180 ry 0 rz -11.91 deg; joints [28.636, -39.771, 104.068, -74.594, 96.848, 154.415]
  MoveL 1114 to (216.75, 49.11, -7.47) mm, rotated rx 180 ry 0 rz -11.91 deg; joints [28.635, -39.766, 104.055, -74.596, 96.849, 154.408]
  MoveL 1115 to (216.79, 49.24, -7.48) mm, rotated rx 180 ry 0 rz -11.91 deg; joints [28.633, -39.76, 104.043, -74.598, 96.851, 154.401]
  MoveL 1116 to (216.84, 49.48, -7.48) mm, rotated rx 180 ry 0 rz -11.91 deg; joints [28.63, -39.751, 104.021, -74.602, 96.853, 154.388]
  MoveL 1117 to (216.87, 49.73, -7.47) mm, rotated rx -180 ry 0 rz -11.91 deg; joints [28.627, -39.742, 104, -74.606, 96.855, 154.376]
  MoveL 1118 to (216.88, 49.97, -7.47) mm, rotated rx -180 ry 0 rz -11.91 deg; joints [28.623, -39.733, 103.98, -74.611, 96.856, 154.365]
  MoveL 1119 to (216.87, 50.21, -7.48) mm, rotated rx 180 ry 0 rz -11.91 deg; joints [28.618, -39.725, 103.961, -74.617, 96.857, 154.354]
  MoveL 1120 to (216.85, 50.45, -7.48) mm, rotated rx -180 ry 0 rz -11.91 deg; joints [28.613, -39.716, 103.942, -74.623, 96.857, 154.343]
  MoveL 1121 to (216.8, 50.69, -7.48) mm, rotated rx 180 ry 0 rz -11.91 deg; joints [28.607, -39.709, 103.924, -74.629, 96.857, 154.333]
  MoveL 1122 to (216.74, 50.93, -7.47) mm, rotated rx 180 ry 0 rz -11.91 deg; joints [28.6, -39.701, 103.908, -74.637, 96.857, 154.323]
  MoveL 1123 to (216.65, 51.17, -7.48) mm, rotated rx 180 ry 0 rz -11.91 deg; joints [28.593, -39.694, 103.892, -74.644, 96.856, 154.313]
  MoveL 1124 to (216.58, 51.34, -7.47) mm, rotated rx 180 ry 0 rz -11.91 deg; joints [28.588, -39.69, 103.882, -74.65, 96.856, 154.307]
  MoveL 1125 to (216.5, 51.5, -7.48) mm, rotated rx 180 ry 0 rz -11.91 deg; joints [28.582, -39.686, 103.872, -74.656, 96.855, 154.301]
  MoveL 1126 to (216.41, 51.67, -7.48) mm, rotated rx -180 ry 0 rz -11.91 deg; joints [28.576, -39.681, 103.863, -74.662, 96.853, 154.296]
  MoveL 1127 to (216.3, 51.83, -7.48) mm, rotated rx -180 ry 0 rz -11.91 deg; joints [28.569, -39.678, 103.854, -74.669, 96.852, 154.29]
  MoveL 1128 to (216.2, 51.96, -7.48) mm, rotated rx -180 ry 0 rz -11.91 deg; joints [28.563, -39.675, 103.848, -74.674, 96.85, 154.286]
  MoveL 1129 to (216.09, 52.1, -7.48) mm, rotated rx -180 ry 0 rz -11.91 deg; joints [28.557, -39.672, 103.842, -74.681, 96.849, 154.282]
  MoveL 1130 to (215.96, 52.23, -7.48) mm, rotated rx 180 ry 0 rz -11.91 deg; joints [28.55, -39.67, 103.836, -74.687, 96.847, 154.278]
  MoveL 1131 to (215.82, 52.37, -7.48) mm, rotated rx 180 ry 0 rz -11.91 deg; joints [28.543, -39.667, 103.832, -74.694, 96.844, 154.275]
  MoveL 1132 to (215.58, 52.56, -7.47) mm, rotated rx -180 ry 0 rz -11.91 deg; joints [28.531, -39.665, 103.826, -74.705, 96.84, 154.271]
  MoveL 1133 to (215.34, 52.72, -7.48) mm, rotated rx -180 ry 0 rz -11.91 deg; joints [28.52, -39.664, 103.824, -74.715, 96.836, 154.269]
  MoveL 1134 to (215.09, 52.85, -7.48) mm, rotated rx -180 ry 0 rz -11.91 deg; joints [28.51, -39.664, 103.824, -74.725, 96.831, 154.268]
  MoveL 1135 to (214.85, 52.96, -7.48) mm, rotated rx 180 ry 0 rz -11.91 deg; joints [28.5, -39.665, 103.826, -74.734, 96.827, 154.268]
  MoveL 1136 to (214.61, 53.04, -7.47) mm, rotated rx 180 ry 0 rz -11.91 deg; joints [28.49, -39.666, 103.83, -74.742, 96.822, 154.269]
  MoveL 1137 to (214.37, 53.1, -7.48) mm, rotated rx -180 ry 0 rz -11.91 deg; joints [28.481, -39.668, 103.836, -74.751, 96.817, 154.271]
  MoveL 1138 to (214.36, 53.11, -7.48) mm, rotated rx 180 ry 0 rz -11.91 deg; joints [28.48, -39.669, 103.836, -74.751, 96.817, 154.271]
  MoveL 1139 to (214.12, 53.15, -7.48) mm, rotated rx -180 ry 0 rz -11.91 deg; joints [28.471, -39.672, 103.843, -74.759, 96.812, 154.274]
  MoveL 1140 to (213.88, 53.17, -7.47) mm, rotated rx -180 ry 0 rz -11.91 deg; joints [28.463, -39.675, 103.852, -74.766, 96.807, 154.278]
  MoveL 1141 to (213.4, 53.17, -7.48) mm, rotated rx 180 ry 0 rz -11.91 deg; joints [28.447, -39.684, 103.873, -74.779, 96.797, 154.288]
  MoveL 1142 to (-195.12, 53.17, -7.48) mm, rotated rx -180 ry 0 rz -11.91 deg; joints [12.975, -44.917, 116.757, -88.773, 89.983, 160.975]
  MoveL 1143 to (-195.28, 53.17, -7.47) mm, rotated rx -180 ry 0 rz -11.91 deg; joints [12.968, -44.918, 116.76, -88.779, 89.981, 160.977]
  MoveL 1144 to (-195.43, 53.16, -7.48) mm, rotated rx 180 ry 0 rz -11.91 deg; joints [12.962, -44.92, 116.764, -88.785, 89.979, 160.98]
  MoveL 1145 to (-195.59, 53.14, -7.47) mm, rotated rx -180 ry 0 rz -11.91 deg; joints [12.956, -44.922, 116.769, -88.791, 89.977, 160.982]
  MoveL 1146 to (-195.75, 53.11, -7.48) mm, rotated rx 180 ry 0 rz -11.91 deg; joints [12.949, -44.924, 116.774, -88.797, 89.975, 160.986]
  MoveL 1147 to (-195.92, 53.07, -7.48) mm, rotated rx -180 ry 0 rz -11.91 deg; joints [12.943, -44.926, 116.781, -88.804, 89.972, 160.99]
  MoveL 1148 to (-196.08, 53.02, -7.47) mm, rotated rx -180 ry 0 rz -11.91 deg; joints [12.936, -44.929, 116.788, -88.81, 89.97, 160.994]
  MoveL 1149 to (-196.25, 52.96, -7.47) mm, rotated rx -180 ry 0 rz -11.91 deg; joints [12.93, -44.932, 116.796, -88.816, 89.968, 160.999]
  MoveL 1150 to (-196.42, 52.89, -7.48) mm, rotated rx 180 ry 0 rz -11.91 deg; joints [12.924, -44.936, 116.805, -88.822, 89.966, 161.004]
  MoveL 1151 to (-196.56, 52.82, -7.47) mm, rotated rx 180 ry 0 rz -11.91 deg; joints [12.919, -44.939, 116.813, -88.827, 89.964, 161.009]
  MoveL 1152 to (-196.7, 52.74, -7.47) mm, rotated rx -180 ry 0 rz -11.91 deg; joints [12.914, -44.943, 116.822, -88.831, 89.963, 161.014]
  MoveL 1153 to (-196.84, 52.66, -7.48) mm, rotated rx 180 ry 0 rz -11.91 deg; joints [12.909, -44.947, 116.832, -88.836, 89.961, 161.02]
  MoveL 1154 to (-196.98, 52.56, -7.48) mm, rotated rx -180 ry 0 rz -11.91 deg; joints [12.904, -44.951, 116.842, -88.841, 89.959, 161.026]
  MoveL 1155 to (-197.12, 52.45, -7.47) mm, rotated rx 180 ry 0 rz -11.91 deg; joints [12.899, -44.956, 116.854, -88.845, 89.958, 161.033]
  MoveL 1156 to (-197.26, 52.33, -7.48) mm, rotated rx 180 ry 0 rz -11.91 deg; joints [12.894, -44.961, 116.867, -88.85, 89.956, 161.041]
  MoveL 1157 to (-197.41, 52.18, -7.48) mm, rotated rx -180 ry 0 rz -11.91 deg; joints [12.889, -44.967, 116.882, -88.854, 89.955, 161.05]
  MoveL 1158 to (-197.54, 52.03, -7.48) mm, rotated rx -180 ry 0 rz -11.91 deg; joints [12.885, -44.973, 116.896, -88.858, 89.953, 161.059]
  MoveL 1159 to (-197.7, 51.82, -7.47) mm, rotated rx -180 ry 0 rz -11.91 deg; joints [12.881, -44.981, 116.917, -88.863, 89.951, 161.071]
  MoveL 1160 to (-197.84, 51.6, -7.48) mm, rotated rx 180 ry 0 rz -11.91 deg; joints [12.877, -44.989, 116.937, -88.866, 89.95, 161.083]
  MoveL 1161 to (-197.95, 51.39, -7.47) mm, rotated rx -180 ry 0 rz -11.91 deg; joints [12.874, -44.997, 116.957, -88.869, 89.949, 161.095]
  MoveL 1162 to (-198.05, 51.18, -7.47) mm, rotated rx 180 ry 0 rz -11.91 deg; joints [12.872, -45.005, 116.976, -88.871, 89.948, 161.106]
  MoveL 1163 to (-198.13, 50.93, -7.47) mm, rotated rx -180 ry 0 rz -11.91 deg; joints [12.871, -45.014, 116.998, -88.872, 89.948, 161.119]
  MoveL 1164 to (-198.2, 50.69, -7.47) mm, rotated rx -180 ry 0 rz -11.91 deg; joints [12.871, -45.022, 117.019, -88.872, 89.947, 161.131]
  MoveL 1165 to (-198.24, 50.45, -7.48) mm, rotated rx -180 ry 0 rz -11.91 deg; joints [12.871, -45.03, 117.039, -88.872, 89.947, 161.144]
  MoveL 1166 to (-198.27, 50.21, -7.47) mm, rotated rx 180 ry 0 rz -11.91 deg; joints [12.873, -45.039, 117.06, -88.87, 89.947, 161.156]
  MoveL 1167 to (-198.27, 49.97, -7.48) mm, rotated rx 180 ry 0 rz -11.91 deg; joints [12.875, -45.047, 117.079, -88.869, 89.948, 161.168]
  MoveL 1168 to (-198.26, 49.73, -7.47) mm, rotated rx -180 ry 0 rz -11.91 deg; joints [12.877, -45.055, 117.099, -88.866, 89.948, 161.179]
  MoveL 1169 to (-198.23, 49.48, -7.48) mm, rotated rx -180 ry 0 rz -11.91 deg; joints [12.881, -45.062, 117.118, -88.862, 89.949, 161.191]
  MoveL 1170 to (-198.18, 49.24, -7.47) mm, rotated rx 180 ry 0 rz -11.91 deg; joints [12.885, -45.07, 117.137, -88.858, 89.95, 161.202]
  MoveL 1171 to (-198.11, 49, -7.48) mm, rotated rx -180 ry 0 rz -11.91 deg; joints [12.891, -45.078, 117.156, -88.853, 89.952, 161.213]
  MoveL 1172 to (-198.02, 48.76, -7.47) mm, rotated rx -180 ry 0 rz -11.91 deg; joints [12.897, -45.085, 117.174, -88.848, 89.953, 161.224]
  MoveL 1173 to (-197.91, 48.52, -7.47) mm, rotated rx -180 ry 0 rz -11.91 deg; joints [12.904, -45.092, 117.191, -88.841, 89.955, 161.234]
  MoveL 1174 to (-197.76, 48.28, -7.48) mm, rotated rx -180 ry 0 rz -11.91 deg; joints [12.912, -45.099, 117.208, -88.833, 89.958, 161.244]
  MoveL 1175 to (-197.66, 48.13, -7.48) mm, rotated rx -180 ry 0 rz -11.91 deg; joints [12.918, -45.103, 117.219, -88.828, 89.959, 161.25]
  MoveL 1176 to (-197.55, 47.98, -7.47) mm, rotated rx 180 ry 0 rz -11.91 deg; joints [12.924, -45.107, 117.228, -88.822, 89.961, 161.256]
  MoveL 1177 to (-197.42, 47.84, -7.48) mm, rotated rx 180 ry 0 rz -11.91 deg; joints [12.931, -45.111, 117.238, -88.815, 89.963, 161.262]
  MoveL 1178 to (-197.27, 47.69, -7.48) mm, rotated rx -180 ry 0 rz -11.91 deg; joints [12.938, -45.115, 117.247, -88.808, 89.965, 161.267]
  MoveL 1179 to (-197.03, 47.48, -7.47) mm, rotated rx -180 ry 0 rz -11.91 deg; joints [12.95, -45.12, 117.26, -88.797, 89.969, 161.275]
  MoveL 1180 to (-196.78, 47.31, -7.47) mm, rotated rx -180 ry 0 rz -11.91 deg; joints [12.962, -45.124, 117.269, -88.785, 89.972, 161.28]
  MoveL 1181 to (-196.6, 47.2, -7.47) mm, rotated rx -180 ry 0 rz -11.91 deg; joints [12.971, -45.126, 117.274, -88.777, 89.975, 161.283]
  Set speed (38.1 mm/s)
  MoveL 1182 to (-196.37, 46.25, -7.47) mm, rotated rx 180 ry 0 rz -11.91 deg; joints [12.989, -45.156, 117.348, -88.759, 89.98, 161.327]
  MoveL 1183 to (-198.16, 43.86, -7.48) mm, rotated rx -180 ry 0 rz -11.91 deg; joints [12.938, -45.248, 117.577, -88.808, 89.961, 161.464]
  MoveL 1184 to (-198.54, 43.36, -6.84) mm, rotated rx 180 ry 0 rz -11.91 deg; joints [12.927, -45.307, 117.632, -88.819, 89.958, 161.46]
  Set speed (100.0 mm/s)
  MoveL 1185 to (-198.54, 43.36, 24.52) mm, rotated rx -180 ry 0 rz -11.91 deg; joints [12.917, -47.241, 117.905, -88.827, 89.989, 159.799]
  MoveL 1186 to (-195.3, 420.76, 24.52) mm, rotated rx 180 ry 0 rz -11.91 deg; joints [10.169, -31.104, 82.184, -91.03, 88.656, 140.218]
  MoveL 1187 to (-195.3, 420.76, 3.11) mm, rotated rx -180 ry 0 rz -11.91 deg; joints [10.174, -30.117, 82.006, -91.045, 88.674, 141.026]
  Set speed (25.4 mm/s)
  MoveL 1188 to (-195.3, 420.76, -0.84) mm, rotated rx 180 ry 0 rz -11.91 deg; joints [10.174, -29.933, 81.969, -91.048, 88.677, 141.173]
  MoveL 1189 to (-195.48, 421.37, -1.47) mm, rotated rx 180 ry 0 rz -11.91 deg; joints [10.165, -29.873, 81.897, -91.055, 88.671, 141.162]
  Set speed (38.1 mm/s)
  MoveL 1190 to (-195.58, 421.7, -1.48) mm, rotated rx 180 ry 0 rz -11.91 deg; joints [10.16, -29.856, 81.861, -91.059, 88.667, 141.142]
  MoveL 1191 to (-194.97, 422.52, -1.48) mm, rotated rx -180 ry 0 rz -11.91 deg; joints [10.175, -29.808, 81.755, -91.045, 88.675, 141.085]
  Set speed (76.2 mm/s)
  MoveL 1192 to (213.41, 422.52, -1.48) mm, rotated rx -180 ry 0 rz -11.91 deg; joints [22.896, -22.923, 66.762, -81.987, 97.69, 133.548]
  MoveL 1193 to (213.89, 422.53, -1.48) mm, rotated rx 180 ry 0 rz -11.91 deg; joints [22.91, -22.91, 66.734, -81.979, 97.702, 133.535]
  MoveL 1194 to (214.13, 422.55, -1.48) mm, rotated rx 180 ry 0 rz -11.91 deg; joints [22.917, -22.903, 66.718, -81.976, 97.708, 133.527]
  MoveL 1195 to (214.37, 422.59, -1.47) mm, rotated rx -180 ry 0 rz -11.91 deg; joints [22.923, -22.894, 66.699, -81.972, 97.714, 133.517]
  MoveL 1196 to (214.61, 422.65, -1.47) mm, rotated rx 180 ry 0 rz -11.91 deg; joints [22.929, -22.883, 66.677, -81.969, 97.72, 133.507]
  MoveL 1197 to (214.85, 422.74, -1.48) mm, rotated rx 180 ry 0 rz -11.91 deg; joints [22.935, -22.872, 66.653, -81.967, 97.726, 133.494]
  MoveL 1198 to (215.09, 422.84, -1.48) mm, rotated rx -180 ry 0 rz -11.91 deg; joints [22.941, -22.859, 66.625, -81.965, 97.732, 133.48]
  MoveL 1199 to (215.34, 422.97, -1.47) mm, rotated rx -180 ry 0 rz -11.91 deg; joints [22.946, -22.845, 66.595, -81.963, 97.738, 133.465]
  MoveL 1200 to (215.58, 423.13, -1.48) mm, rotated rx 180 ry 0 rz -11.91 deg; joints [22.951, -22.828, 66.56, -81.962, 97.744, 133.447]
  MoveL 1201 to (215.82, 423.33, -1.48) mm, rotated rx 180 ry 0 rz -11.91 deg; joints [22.956, -22.81, 66.521, -81.962, 97.751, 133.427]
  MoveL 1202 to (215.96, 423.46, -1.47) mm, rotated rx 180 ry 0 rz -11.91 deg; joints [22.958, -22.798, 66.495, -81.962, 97.754, 133.413]
  MoveL 1203 to (216.09, 423.6, -1.47) mm, rotated rx -180 ry 0 rz -11.91 deg; joints [22.96, -22.786, 66.47, -81.962, 97.758, 133.4]
  MoveL 1204 to (216.2, 423.73, -1.47) mm, rotated rx -180 ry 0 rz -11.91 deg; joints [22.962, -22.775, 66.446, -81.963, 97.76, 133.388]
  MoveL 1205 to (216.3, 423.87, -1.48) mm, rotated rx 180 ry 0 rz -11.91 deg; joints [22.963, -22.763, 66.422, -81.964, 97.763, 133.376]
  MoveL 1206 to (216.39, 424.01, -1.48) mm, rotated rx -180 ry 0 rz -11.91 deg; joints [22.964, -22.752, 66.399, -81.965, 97.765, 133.363]
  MoveL 1207 to (216.47, 424.15, -1.47) mm, rotated rx -180 ry 0 rz -11.91 deg; joints [22.965, -22.741, 66.376, -81.966, 97.768, 133.351]
  MoveL 1208 to (216.6, 424.39, -1.48) mm, rotated rx -180 ry 0 rz -11.91 deg; joints [22.965, -22.723, 66.337, -81.968, 97.771, 133.331]
  MoveL 1209 to (216.69, 424.63, -1.47) mm, rotated rx 180 ry 0 rz -11.91 deg; joints [22.965, -22.705, 66.299, -81.971, 97.774, 133.311]
  MoveL 1210 to (216.77, 424.87, -1.48) mm, rotated rx -180 ry 0 rz -11.91 deg; joints [22.964, -22.688, 66.263, -81.974, 97.776, 133.292]
  MoveL 1211 to (216.82, 425.11, -1.48) mm, rotated rx 180 ry 0 rz -11.91 deg; joints [22.963, -22.671, 66.228, -81.978, 97.777, 133.273]
  MoveL 1212 to (216.86, 425.35, -1.47) mm, rotated rx -180 ry 0 rz -11.91 deg; joints [22.961, -22.655, 66.194, -81.981, 97.778, 133.255]
  MoveL 1213 to (216.88, 425.59, -1.47) mm, rotated rx -180 ry 0 rz -11.91 deg; joints [22.959, -22.64, 66.161, -81.986, 97.779, 133.237]
  MoveL 1214 to (216.88, 425.84, -1.47) mm, rotated rx 180 ry 0 rz -11.91 deg; joints [22.956, -22.624, 66.129, -81.99, 97.779, 133.22]
  MoveL 1215 to (216.87, 426.08, -1.48) mm, rotated rx -180 ry 0 rz -11.91 deg; joints [22.953, -22.609, 66.097, -81.994, 97.779, 133.203]
  MoveL 1216 to (216.85, 426.28, -1.48) mm, rotated rx 180 ry 0 rz -11.91 deg; joints [22.95, -22.597, 66.071, -81.998, 97.779, 133.189]
  MoveL 1217 to (216.82, 426.49, -1.48) mm, rotated rx -180 ry 0 rz -11.91 deg; joints [22.946, -22.585, 66.046, -82.003, 97.778, 133.176]
  MoveL 1218 to (216.77, 426.69, -1.48) mm, rotated rx 180 ry 0 rz -11.91 deg; joints [22.942, -22.573, 66.021, -82.007, 97.777, 133.162]
  MoveL 1219 to (216.71, 426.89, -1.48) mm, rotated rx 180 ry 0 rz -11.91 deg; joints [22.938, -22.562, 65.997, -82.012, 97.776, 133.15]
  MoveL 1220 to (216.64, 427.1, -1.47) mm, rotated rx -180 ry 0 rz -11.91 deg; joints [22.933, -22.551, 65.974, -82.017, 97.774, 133.137]
  MoveL 1221 to (216.54, 427.3, -1.48) mm, rotated rx 180 ry 0 rz -11.91 deg; joints [22.928, -22.541, 65.953, -82.022, 97.772, 133.125]
  MoveL 1222 to (216.43, 427.51, -1.47) mm, rotated rx -180 ry 0 rz -11.91 deg; joints [22.922, -22.531, 65.932, -82.027, 97.77, 133.114]
  MoveL 1223 to (216.3, 427.71, -1.48) mm, rotated rx 180 ry 0 rz -11.91 deg; joints [22.916, -22.521, 65.912, -82.033, 97.767, 133.103]
  MoveL 1224 to (216.19, 427.86, -1.47) mm, rotated rx -180 ry 0 rz -11.91 deg; joints [22.911, -22.515, 65.898, -82.038, 97.764, 133.095]
  MoveL 1225 to (216.06, 428.01, -1.47) mm, rotated rx 180 ry 0 rz -11.91 deg; joints [22.905, -22.509, 65.885, -82.042, 97.761, 133.088]
  MoveL 1226 to (215.85, 428.22, -1.48) mm, rotated rx -180 ry 0 rz -11.91 deg; joints [22.897, -22.501, 65.869, -82.05, 97.756, 133.078]
  MoveL 1227 to (215.64, 428.4, -1.48) mm, rotated rx 180 ry 0 rz -11.91 deg; joints [22.889, -22.495, 65.857, -82.056, 97.751, 133.071]
  MoveL 1228 to (215.43, 428.55, -1.47) mm, rotated rx 180 ry 0 rz -11.91 deg; joints [22.881, -22.491, 65.849, -82.062, 97.746, 133.066]
  MoveL 1229 to (215.21, 428.67, -1.48) mm, rotated rx 180 ry 0 rz -11.91 deg; joints [22.873, -22.489, 65.845, -82.068, 97.74, 133.063]
  MoveL 1230 to (215, 428.78, -1.48) mm, rotated rx -180 ry 0 rz -11.91 deg; joints [22.866, -22.488, 65.843, -82.073, 97.735, 133.062]
  MoveL 1231 to (214.79, 428.86, -1.48) mm, rotated rx 180 ry 0 rz -11.91 deg; joints [22.859, -22.488, 65.843, -82.078, 97.73, 133.061]
  MoveL 1232 to (214.58, 428.93, -1.48) mm, rotated rx 180 ry 0 rz -11.91 deg; joints [22.852, -22.489, 65.846, -82.083, 97.725, 133.062]
  MoveL 1233 to (214.37, 428.98, -1.48) mm, rotated rx 180 ry 0 rz -11.91 deg; joints [22.845, -22.491, 65.851, -82.087, 97.72, 133.064]
  MoveL 1234 to (214.13, 429.03, -1.48) mm, rotated rx -180 ry 0 rz -11.91 deg; joints [22.837, -22.495, 65.859, -82.092, 97.714, 133.067]
  MoveL 1235 to (213.89, 429.05, -1.48) mm, rotated rx 180 ry 0 rz -11.91 deg; joints [22.83, -22.5, 65.869, -82.096, 97.708, 133.072]
  MoveL 1236 to (213.41, 429.06, -1.48) mm, rotated rx 180 ry 0 rz -11.91 deg; joints [22.816, -22.512, 65.895, -82.104, 97.696, 133.085]
  MoveL 1237 to (-194.97, 429.06, -1.48) mm, rotated rx -180 ry 0 rz -11.91 deg; joints [10.136, -29.461, 81.007, -91.067, 88.644, 140.684]
  MoveL 1238 to (-195.21, 429.05, -1.47) mm, rotated rx -180 ry 0 rz -11.91 deg; joints [10.128, -29.464, 81.012, -91.073, 88.639, 140.687]
  MoveL 1239 to (-195.45, 429.04, -1.48) mm, rotated rx -180 ry 0 rz -11.91 deg; joints [10.12, -29.467, 81.019, -91.079, 88.634, 140.691]
  MoveL 1240 to (-195.69, 429, -1.48) mm, rotated rx -180 ry 0 rz -11.91 deg; joints [10.112, -29.471, 81.028, -91.085, 88.629, 140.696]
  MoveL 1241 to (-195.93, 428.94, -1.47) mm, rotated rx 180 ry 0 rz -11.91 deg; joints [10.105, -29.476, 81.04, -91.091, 88.625, 140.702]
  MoveL 1242 to (-196.18, 428.87, -1.48) mm, rotated rx -180 ry 0 rz -11.91 deg; joints [10.097, -29.483, 81.053, -91.097, 88.62, 140.71]
  MoveL 1243 to (-196.42, 428.77, -1.48) mm, rotated rx -180 ry 0 rz -11.91 deg; joints [10.09, -29.49, 81.07, -91.103, 88.616, 140.718]
  MoveL 1244 to (-196.55, 428.71, -1.48) mm, rotated rx -180 ry 0 rz -11.91 deg; joints [10.086, -29.495, 81.079, -91.107, 88.614, 140.724]
  MoveL 1245 to (-196.68, 428.64, -1.47) mm, rotated rx -180 ry 0 rz -11.91 deg; joints [10.082, -29.5, 81.09, -91.11, 88.611, 140.73]
  MoveL 1246 to (-196.81, 428.56, -1.48) mm, rotated rx 180 ry 0 rz -11.91 deg; joints [10.078, -29.505, 81.102, -91.113, 88.609, 140.736]
  MoveL 1247 to (-196.93, 428.47, -1.48) mm, rotated rx -180 ry 0 rz -11.91 deg; joints [10.075, -29.511, 81.115, -91.116, 88.607, 140.743]
  MoveL 1248 to (-197.06, 428.37, -1.48) mm, rotated rx -180 ry 0 rz -11.91 deg; joints [10.071, -29.517, 81.128, -91.119, 88.605, 140.75]
  MoveL 1249 to (-197.19, 428.27, -1.48) mm, rotated rx -180 ry 0 rz -11.91 deg; joints [10.067, -29.524, 81.143, -91.122, 88.603, 140.759]
  MoveL 1250 to (-197.32, 428.15, -1.47) mm, rotated rx -180 ry 0 rz -11.91 deg; joints [10.064, -29.532, 81.16, -91.125, 88.601, 140.767]
  MoveL 1251 to (-197.45, 428.01, -1.47) mm, rotated rx 180 ry 0 rz -11.91 deg; joints [10.06, -29.54, 81.178, -91.128, 88.599, 140.777]
  MoveL 1252 to (-197.65, 427.77, -1.48) mm, rotated rx -180 ry 0 rz -11.91 deg; joints [10.055, -29.555, 81.21, -91.132, 88.596, 140.794]
  MoveL 1253 to (-197.81, 427.53, -1.47) mm, rotated rx -180 ry 0 rz -11.91 deg; joints [10.051, -29.569, 81.241, -91.136, 88.594, 140.811]
  MoveL 1254 to (-197.94, 427.29, -1.48) mm, rotated rx -180 ry 0 rz -11.91 deg; joints [10.048, -29.583, 81.271, -91.139, 88.592, 140.828]
  MoveL 1255 to (-198.05, 427.04, -1.48) mm, rotated rx -180 ry 0 rz -11.91 deg; joints [10.046, -29.597, 81.301, -91.141, 88.591, 140.844]
  MoveL 1256 to (-198.14, 426.8, -1.47) mm, rotated rx 180 ry 0 rz -11.91 deg; joints [10.045, -29.61, 81.331, -91.142, 88.591, 140.86]
  MoveL 1257 to (-198.2, 426.56, -1.48) mm, rotated rx -180 ry 0 rz -11.91 deg; joints [10.044, -29.624, 81.36, -91.143, 88.591, 140.875]
  MoveL 1258 to (-198.24, 426.32, -1.48) mm, rotated rx 180 ry 0 rz -11.91 deg; joints [10.044, -29.637, 81.388, -91.143, 88.591, 140.891]
  MoveL 1259 to (-198.27, 426.08, -1.47) mm, rotated rx -180 ry 0 rz -11.91 deg; joints [10.045, -29.65, 81.416, -91.143, 88.592, 140.906]
  MoveL 1260 to (-198.27, 425.84, -1.48) mm, rotated rx -180 ry 0 rz -11.91 deg; joints [10.046, -29.663, 81.444, -91.143, 88.593, 140.921]
  MoveL 1261 to (-198.27, 425.59, -1.48) mm, rotated rx -180 ry 0 rz -11.91 deg; joints [10.048, -29.676, 81.472, -91.142, 88.594, 140.935]
  MoveL 1262 to (-198.25, 425.35, -1.48) mm, rotated rx 180 ry 0 rz -11.91 deg; joints [10.05, -29.688, 81.499, -91.141, 88.595, 140.95]
  MoveL 1263 to (-198.22, 425.11, -1.48) mm, rotated rx -180 ry 0 rz -11.91 deg; joints [10.052, -29.701, 81.526, -91.139, 88.597, 140.964]
  MoveL 1264 to (-198.16, 424.87, -1.48) mm, rotated rx -180 ry 0 rz -11.91 deg; joints [10.055, -29.713, 81.552, -91.137, 88.6, 140.979]
  MoveL 1265 to (-198.09, 424.63, -1.48) mm, rotated rx -180 ry 0 rz -11.91 deg; joints [10.059, -29.725, 81.578, -91.134, 88.602, 140.993]
  MoveL 1266 to (-197.99, 424.39, -1.47) mm, rotated rx -180 ry 0 rz -11.91 deg; joints [10.064, -29.737, 81.604, -91.131, 88.605, 141.006]
  MoveL 1267 to (-197.87, 424.15, -1.47) mm, rotated rx 180 ry 0 rz -11.91 deg; joints [10.069, -29.749, 81.629, -91.127, 88.609, 141.02]
  MoveL 1268 to (-197.73, 423.93, -1.48) mm, rotated rx 180 ry 0 rz -11.91 deg; joints [10.075, -29.759, 81.651, -91.123, 88.613, 141.032]
  MoveL 1269 to (-197.57, 423.71, -1.47) mm, rotated rx -180 ry 0 rz -11.91 deg; joints [10.082, -29.769, 81.673, -91.118, 88.617, 141.043]
  MoveL 1270 to (-197.38, 423.49, -1.48) mm, rotated rx 180 ry 0 rz -11.91 deg; joints [10.09, -29.779, 81.694, -91.112, 88.622, 141.054]
  MoveL 1271 to (-197.14, 423.27, -1.47) mm, rotated rx -180 ry 0 rz -11.91 deg; joints [10.099, -29.788, 81.715, -91.105, 88.628, 141.065]
  MoveL 1272 to (-196.96, 423.13, -1.47) mm, rotated rx -180 ry 0 rz -11.91 deg; joints [10.105, -29.794, 81.727, -91.1, 88.632, 141.072]
  MoveL 1273 to (-196.78, 423, -1.47) mm, rotated rx -180 ry 0 rz -11.91 deg; joints [10.112, -29.799, 81.737, -91.095, 88.637, 141.077]
  MoveL 1274 to (-196.6, 422.9, -1.47) mm, rotated rx -180 ry 0 rz -11.91 deg; joints [10.119, -29.803, 81.745, -91.089, 88.641, 141.081]
  MoveL 1275 to (-196.42, 422.81, -1.47) mm, rotated rx 180 ry 0 rz -11.91 deg; joints [10.125, -29.806, 81.752, -91.084, 88.645, 141.085]
  MoveL 1276 to (-196.18, 422.71, -1.48) mm, rotated rx -180 ry 0 rz -11.91 deg; joints [10.134, -29.809, 81.758, -91.078, 88.65, 141.088]
  MoveL 1277 to (-195.93, 422.63, -1.47) mm, rotated rx -180 ry 0 rz -11.91 deg; joints [10.142, -29.811, 81.762, -91.071, 88.655, 141.09]
  MoveL 1278 to (-195.69, 422.58, -1.47) mm, rotated rx 180 ry 0 rz -11.91 deg; joints [10.151, -29.811, 81.763, -91.065, 88.66, 141.09]
  MoveL 1279 to (-195.45, 422.54, -1.48) mm, rotated rx 180 ry 0 rz -11.91 deg; joints [10.159, -29.811, 81.763, -91.058, 88.666, 141.09]
  MoveL 1280 to (-195.21, 422.52, -1.47) mm, rotated rx 180 ry 0 rz -11.91 deg; joints [10.167, -29.81, 81.76, -91.052, 88.67, 141.088]
  MoveL 1281 to (-194.97, 422.52, -1.48) mm, rotated rx -180 ry 0 rz -11.91 deg; joints [10.175, -29.808, 81.755, -91.045, 88.675, 141.085]
  Set speed (38.1 mm/s)
  MoveL 1282 to (-194.97, 421.25, -1.47) mm, rotated rx -180 ry 0 rz -11.91 deg; joints [10.182, -29.875, 81.9, -91.041, 88.681, 141.163]
  MoveL 1283 to (-195.61, 421.25, -1.47) mm, rotated rx -180 ry 0 rz -11.91 deg; joints [10.161, -29.881, 81.913, -91.058, 88.669, 141.17]
  Set speed (25.4 mm/s)
  MoveL 1284 to (-195.61, 421.25, -3.84) mm, rotated rx 180 ry 0 rz -11.91 deg; joints [10.162, -29.77, 81.89, -91.06, 88.671, 141.258]
  MoveL 1285 to (-195.61, 421.89, -4.47) mm, rotated rx -180 ry 0 rz -11.91 deg; joints [10.158, -29.707, 81.811, -91.062, 88.668, 141.242]
  Set speed (38.1 mm/s)
  MoveL 1286 to (-194.97, 422.52, -4.47) mm, rotated rx -180 ry 0 rz -11.91 deg; joints [10.175, -29.668, 81.726, -91.047, 88.678, 141.196]
  Set speed (76.2 mm/s)
  MoveL 1287 to (213.41, 422.52, -4.47) mm, rotated rx -180 ry 0 rz -11.91 deg; joints [22.897, -22.791, 66.729, -81.973, 97.677, 133.647]
  MoveL 1288 to (213.89, 422.53, -4.48) mm, rotated rx 180 ry 0 rz -11.91 deg; joints [22.911, -22.778, 66.701, -81.965, 97.689, 133.634]
  MoveL 1289 to (214.13, 422.55, -4.47) mm, rotated rx -180 ry 0 rz -11.91 deg; joints [22.918, -22.771, 66.685, -81.962, 97.695, 133.626]
  MoveL 1290 to (214.37, 422.59, -4.47) mm, rotated rx -180 ry 0 rz -11.91 deg; joints [22.924, -22.762, 66.666, -81.958, 97.701, 133.616]
  MoveL 1291 to (214.61, 422.65, -4.48) mm, rotated rx 180 ry 0 rz -11.91 deg; joints [22.93, -22.751, 66.644, -81.956, 97.707, 133.606]
  MoveL 1292 to (214.85, 422.74, -4.48) mm, rotated rx -180 ry 0 rz -11.91 deg; joints [22.936, -22.74, 66.62, -81.953, 97.713, 133.593]
  MoveL 1293 to (215.09, 422.84, -4.48) mm, rotated rx 180 ry 0 rz -11.91 deg; joints [22.942, -22.727, 66.592, -81.951, 97.719, 133.579]
  MoveL 1294 to (215.34, 422.97, -4.48) mm, rotated rx -180 ry 0 rz -11.91 deg; joints [22.947, -22.713, 66.561, -81.949, 97.725, 133.564]
  MoveL 1295 to (215.58, 423.13, -4.47) mm, rotated rx -180 ry 0 rz -11.91 deg; joints [22.952, -22.696, 66.527, -81.948, 97.731, 133.546]
  MoveL 1296 to (215.82, 423.33, -4.47) mm, rotated rx -180 ry 0 rz -11.91 deg; joints [22.957, -22.678, 66.488, -81.948, 97.737, 133.526]
  MoveL 1297 to (215.96, 423.46, -4.47) mm, rotated rx -180 ry 0 rz -11.91 deg; joints [22.959, -22.666, 66.462, -81.948, 97.741, 133.512]
  MoveL 1298 to (216.09, 423.6, -4.48) mm, rotated rx -180 ry 0 rz -11.91 deg; joints [22.961, -22.654, 66.437, -81.948, 97.744, 133.499]
  MoveL 1299 to (216.2, 423.73, -4.47) mm, rotated rx -180 ry 0 rz -11.91 deg; joints [22.963, -22.643, 66.413, -81.949, 97.747, 133.487]
  MoveL 1300 to (216.3, 423.87, -4.47) mm, rotated rx -180 ry 0 rz -11.91 deg; joints [22.964, -22.631, 66.389, -81.95, 97.75, 133.474]
  MoveL 1301 to (216.39, 424.01, -4.47) mm, rotated rx -180 ry 0 rz -11.91 deg; joints [22.965, -22.62, 66.366, -81.951, 97.752, 133.462]
  MoveL 1302 to (216.47, 424.15, -4.48) mm, rotated rx 180 ry 0 rz -11.91 deg; joints [22.966, -22.61, 66.343, -81.952, 97.755, 133.45]
  MoveL 1303 to (216.6, 424.39, -4.47) mm, rotated rx -180 ry 0 rz -11.91 deg; joints [22.966, -22.591, 66.304, -81.954, 97.758, 133.429]
  MoveL 1304 to (216.69, 424.63, -4.48) mm, rotated rx -180 ry 0 rz -11.91 deg; joints [22.966, -22.573, 66.266, -81.957, 97.76, 133.41]
  MoveL 1305 to (216.77, 424.87, -4.48) mm, rotated rx 180 ry 0 rz -11.91 deg; joints [22.965, -22.556, 66.23, -81.96, 97.763, 133.39]
  MoveL 1306 to (216.82, 425.11, -4.48) mm, rotated rx 180 ry 0 rz -11.91 deg; joints [22.964, -22.54, 66.195, -81.964, 97.764, 133.372]
  MoveL 1307 to (216.86, 425.35, -4.48) mm, rotated rx -180 ry 0 rz -11.91 deg; joints [22.962, -22.523, 66.161, -81.968, 97.765, 133.354]
  MoveL 1308 to (216.88, 425.59, -4.48) mm, rotated rx -180 ry 0 rz -11.91 deg; joints [22.96, -22.508, 66.128, -81.972, 97.766, 133.336]
  MoveL 1309 to (216.88, 426.08, -4.48) mm, rotated rx 180 ry 0 rz -11.91 deg; joints [22.954, -22.477, 66.063, -81.98, 97.766, 133.302]
  MoveL 1310 to (216.88, 426.56, -4.48) mm, rotated rx -180 ry 0 rz -11.91 deg; joints [22.948, -22.447, 65.999, -81.989, 97.767, 133.267]
  MoveL 1311 to (216.86, 426.8, -4.48) mm, rotated rx -180 ry 0 rz -11.91 deg; joints [22.944, -22.432, 65.968, -81.994, 97.767, 133.251]
  MoveL 1312 to (216.82, 427.04, -4.48) mm, rotated rx 180 ry 0 rz -11.91 deg; joints [22.94, -22.418, 65.938, -81.999, 97.766, 133.234]
  MoveL 1313 to (216.76, 427.29, -4.48) mm, rotated rx -180 ry 0 rz -11.91 deg; joints [22.935, -22.404, 65.909, -82.004, 97.765, 133.219]
  MoveL 1314 to (216.68, 427.53, -4.47) mm, rotated rx -180 ry 0 rz -11.91 deg; joints [22.93, -22.391, 65.881, -82.01, 97.763, 133.204]
  MoveL 1315 to (216.58, 427.77, -4.48) mm, rotated rx 180 ry 0 rz -11.91 deg; joints [22.924, -22.378, 65.855, -82.016, 97.761, 133.189]
  MoveL 1316 to (216.46, 428.01, -4.47) mm, rotated rx 180 ry 0 rz -11.91 deg; joints [22.918, -22.366, 65.829, -82.022, 97.758, 133.175]
  MoveL 1317 to (216.3, 428.26, -4.48) mm, rotated rx 180 ry 0 rz -11.91 deg; joints [22.91, -22.355, 65.805, -82.029, 97.754, 133.162]
  MoveL 1318 to (216.2, 428.39, -4.48) mm, rotated rx -180 ry 0 rz -11.91 deg; joints [22.906, -22.349, 65.793, -82.033, 97.752, 133.155]
  MoveL 1319 to (216.09, 428.53, -4.47) mm, rotated rx -180 ry 0 rz -11.91 deg; joints [22.901, -22.343, 65.781, -82.037, 97.749, 133.148]
  MoveL 1320 to (215.96, 428.66, -4.48) mm, rotated rx 180 ry 0 rz -11.91 deg; joints [22.896, -22.338, 65.77, -82.042, 97.746, 133.142]
  MoveL 1321 to (215.82, 428.8, -4.48) mm, rotated rx -180 ry 0 rz -11.91 deg; joints [22.89, -22.333, 65.76, -82.047, 97.743, 133.136]
  MoveL 1322 to (215.58, 428.99, -4.47) mm, rotated rx 180 ry 0 rz -11.91 deg; joints [22.88, -22.327, 65.748, -82.054, 97.737, 133.129]
  MoveL 1323 to (215.34, 429.15, -4.48) mm, rotated rx 180 ry 0 rz -11.91 deg; joints [22.872, -22.324, 65.74, -82.061, 97.731, 133.124]
  MoveL 1324 to (215.09, 429.28, -4.47) mm, rotated rx -180 ry 0 rz -11.91 deg; joints [22.863, -22.322, 65.736, -82.067, 97.725, 133.121]
  MoveL 1325 to (214.85, 429.39, -4.48) mm, rotated rx -180 ry 0 rz -11.91 deg; joints [22.855, -22.321, 65.736, -82.073, 97.719, 133.12]
  MoveL 1326 to (214.61, 429.47, -4.48) mm, rotated rx -180 ry 0 rz -11.91 deg; joints [22.847, -22.322, 65.738, -82.078, 97.713, 133.121]
  MoveL 1327 to (214.37, 429.53, -4.47) mm, rotated rx -180 ry 0 rz -11.91 deg; joints [22.839, -22.325, 65.744, -82.083, 97.707, 133.123]
  MoveL 1328 to (214.13, 429.58, -4.47) mm, rotated rx 180 ry 0 rz -11.91 deg; joints [22.832, -22.329, 65.752, -82.088, 97.701, 133.127]
  MoveL 1329 to (213.89, 429.6, -4.47) mm, rotated rx -180 ry 0 rz -11.91 deg; joints [22.824, -22.333, 65.762, -82.092, 97.695, 133.131]
  MoveL 1330 to (213.41, 429.6, -4.48) mm, rotated rx -180 ry 0 rz -11.91 deg; joints [22.811, -22.346, 65.789, -82.1, 97.683, 133.144]
  MoveL 1331 to (-194.97, 429.6, -4.48) mm, rotated rx 180 ry 0 rz -11.91 deg; joints [10.133, -29.293, 80.914, -91.07, 88.644, 140.76]
  MoveL 1332 to (-195.21, 429.6, -4.47) mm, rotated rx -180 ry 0 rz -11.91 deg; joints [10.125, -29.295, 80.919, -91.077, 88.639, 140.763]
  MoveL 1333 to (-195.45, 429.58, -4.47) mm, rotated rx -180 ry 0 rz -11.91 deg; joints [10.118, -29.298, 80.926, -91.083, 88.634, 140.767]
  MoveL 1334 to (-195.69, 429.55, -4.47) mm, rotated rx 180 ry 0 rz -11.91 deg; joints [10.11, -29.302, 80.936, -91.089, 88.629, 140.772]
  MoveL 1335 to (-195.93, 429.49, -4.48) mm, rotated rx 180 ry 0 rz -11.91 deg; joints [10.102, -29.308, 80.947, -91.095, 88.625, 140.778]
  MoveL 1336 to (-196.18, 429.42, -4.47) mm, rotated rx -180 ry 0 rz -11.91 deg; joints [10.095, -29.314, 80.961, -91.101, 88.62, 140.786]
  MoveL 1337 to (-196.42, 429.32, -4.47) mm, rotated rx 180 ry 0 rz -11.91 deg; joints [10.087, -29.321, 80.977, -91.107, 88.616, 140.795]
  MoveL 1338 to (-196.6, 429.23, -4.47) mm, rotated rx 180 ry 0 rz -11.91 deg; joints [10.082, -29.328, 80.991, -91.112, 88.613, 140.802]
  MoveL 1339 to (-196.78, 429.13, -4.48) mm, rotated rx -180 ry 0 rz -11.91 deg; joints [10.077, -29.335, 81.007, -91.116, 88.609, 140.811]
  MoveL 1340 to (-196.95, 429.01, -4.47) mm, rotated rx -180 ry 0 rz -11.91 deg; joints [10.072, -29.343, 81.024, -91.12, 88.606, 140.82]
  MoveL 1341 to (-197.13, 428.87, -4.48) mm, rotated rx 180 ry 0 rz -11.91 deg; joints [10.066, -29.352, 81.044, -91.125, 88.604, 140.831]
